  MoveL 9498 to (499.58, 497.3, 18) mm, rotated rx 0 ry 90 rz 0 deg; joints [-11.769, -28.209, 111.796, -15.788, -82.965, 50.97]
  Set speed (15.0 mm/s)
  MoveL 9499 to (498.36, 498.52, 18) mm, rotated rx 0 ry 90 rz 0 deg; joints [-11.905, -28.227, 111.911, -15.921, -83.063, 50.957]
  Set speed (120.0 mm/s)
  MoveL 9500 to (498.02, 497.86, 18) mm, rotated rx 0 ry 90 rz 0 deg; joints [-11.851, -28.235, 111.967, -15.865, -83.107, 50.939]
  Set speed (15.0 mm/s)
  Call Extruder(0.050)
  MoveL 9501 to (499.24, 496.65, 18) mm, rotated rx 0 ry 90 rz 0 deg; joints [-11.715, -28.217, 111.852, -15.733, -83.009, 50.951]
  Set speed (120.0 mm/s)
  MoveL 9502 to (498.91, 495.99, 18) mm, rotated rx 0 ry 90 rz 0 deg; joints [-11.662, -28.226, 111.909, -15.677, -83.053, 50.932]
  Set speed (15.0 mm/s)
  Call Extruder(0.050)
  MoveL 9503 to (497.69, 497.21, 18) mm, rotated rx 0 ry 90 rz 0 deg; joints [-11.797, -28.244, 112.024, -15.81, -83.151, 50.92]
  Set speed (120.0 mm/s)
  MoveL 9504 to (497.36, 496.55, 18) mm, rotated rx 0 ry 90 rz 0 deg; joints [-11.743, -28.253, 112.08, -15.754, -83.195, 50.901]
  Set speed (15.0 mm/s)
  Call Extruder(0.107)
  MoveL 9505 to (499.95, 493.96, 18) mm, rotated rx 0 ry 90 rz 0 deg; joints [-11.455, -28.215, 111.834, -15.471, -82.986, 50.927]
  Set speed (120.0 mm/s)
  MoveL 9506 to (498.96, 493.96, 18) mm, rotated rx 0 ry 90 rz 0 deg; joints [-11.474, -28.233, 111.952, -15.486, -83.083, 50.902]
  Set speed (15.0 mm/s)
  Call Extruder(0.080)
  MoveL 9507 to (497.02, 495.9, 18) mm, rotated rx 0 ry 90 rz 0 deg; joints [-11.689, -28.262, 112.136, -15.698, -83.239, 50.883]
  Set speed (120.0 mm/s)
  MoveL 9508 to (496.69, 495.24, 18) mm, rotated rx 0 ry 90 rz 0 deg; joints [-11.635, -28.27, 112.192, -15.642, -83.283, 50.864]
  Set speed (15.0 mm/s)
  Call Extruder(0.053)
  MoveL 9509 to (497.97, 493.96, 18) mm, rotated rx 0 ry 90 rz 0 deg; joints [-11.492, -28.251, 112.07, -15.502, -83.18, 50.877]
  Set speed (120.0 mm/s)
  MoveL 9510 to (496.98, 493.96, 18) mm, rotated rx 0 ry 90 rz 0 deg; joints [-11.511, -28.27, 112.189, -15.517, -83.277, 50.852]
  Set speed (15.0 mm/s)
  Call Extruder(0.026)
  MoveL 9511 to (496.35, 494.59, 18) mm, rotated rx 0 ry 90 rz 0 deg; joints [-11.58, -28.279, 112.248, -15.586, -83.327, 50.846]
  Set speed (120.0 mm/s)
  MoveL 9512 to (499.33, 495.57, 18) mm, rotated rx 0 ry 90 rz 0 deg; joints [-11.614, -28.22, 111.868, -15.63, -83.019, 50.936]
  Set speed (15.0 mm/s)
  Call Extruder(0.066)
  MoveL 9513 to (500.94, 493.96, 18) mm, rotated rx 0 ry 90 rz 0 deg; joints [-11.437, -28.196, 111.716, -15.456, -82.89, 50.952]
  Set speed (120.0 mm/s)
  MoveL 9514 to (501.93, 493.96, 18) mm, rotated rx 0 ry 90 rz 0 deg; joints [-11.418, -28.177, 111.597, -15.441, -82.793, 50.976]
  Set speed (15.0 mm/s)
  MoveL 9515 to (500.32, 495.57, 18) mm, rotated rx 0 ry 90 rz 0 deg; joints [-11.596, -28.201, 111.75, -15.615, -82.922, 50.961]
  Set speed (120.0 mm/s)
  MoveL 9516 to (501.31, 495.57, 18) mm, rotated rx 0 ry 90 rz 0 deg; joints [-11.577, -28.183, 111.632, -15.599, -82.826, 50.986]
  Set speed (15.0 mm/s)
  MoveL 9517 to (502.92, 493.96, 18) mm, rotated rx 0 ry 90 rz 0 deg; joints [-11.4, -28.158, 111.478, -15.426, -82.697, 51.001]
  Set speed (120.0 mm/s)
  MoveL 9518 to (503.91, 493.96, 18) mm, rotated rx 0 ry 90 rz 0 deg; joints [-11.382, -28.139, 111.36, -15.411, -82.6, 51.026]
  Set speed (15.0 mm/s)
  MoveL 9519 to (502.3, 495.57, 18) mm, rotated rx 0 ry 90 rz 0 deg; joints [-11.558, -28.164, 111.513, -15.584, -82.729, 51.011]
  Set speed (120.0 mm/s)
  MoveL 9520 to (503.29, 495.57, 18) mm, rotated rx 0 ry 90 rz 0 deg; joints [-11.54, -28.144, 111.394, -15.569, -82.633, 51.036]
  Set speed (15.0 mm/s)
  Call Extruder(0.035)
  MoveL 9521 to (504.15, 494.7, 18) mm, rotated rx 0 ry 90 rz 0 deg; joints [-11.445, -28.131, 111.312, -15.476, -82.563, 51.044]
  Set speed (120.0 mm/s)
  MoveL 9522 to (502.26, 502.54, 18) mm, rotated rx 0 ry 90 rz 0 deg; joints [-12.196, -28.136, 111.343, -16.232, -82.613, 51.123]
  Set speed (15.0 mm/s)
  Call Extruder(0.050)
  MoveL 9523 to (501.03, 503.76, 18) mm, rotated rx 0 ry 90 rz 0 deg; joints [-12.332, -28.155, 111.457, -16.365, -82.709, 51.111]
  MoveL 9524 to (500.91, 503.89, 18) mm, rotated rx 0 ry 90 rz 0 deg; joints [-12.346, -28.156, 111.469, -16.379, -82.719, 51.11]
  Set speed (120.0 mm/s)
  MoveL 9525 to (490.68, 490.68, 18) mm, rotated rx 0 ry 90 rz 0 deg; joints [-11.324, -28.393, 113.016, -15.308, -83.95, 50.646]
  Set speed (1000.0 mm/s)
  MoveL 9526 to (490.68, 490.68, 18.1) mm, rotated rx 0 ry 90 rz 0 deg; joints [-11.324, -28.403, 113.021, -15.309, -83.945, 50.647]
  Set speed (30.0 mm/s)
  Call Extruder(0.249)
  MoveL 9527 to (496.74, 496.74, 18.1) mm, rotated rx 0 ry 90 rz 0 deg; joints [-11.772, -28.274, 112.154, -15.781, -83.247, 50.89]
  MoveL 9528 to (496.86, 496.86, 18.1) mm, rotated rx 0 ry 90 rz 0 deg; joints [-11.781, -28.271, 112.137, -15.791, -83.233, 50.895]
  Set speed (120.0 mm/s)
  MoveL 9529 to (495.64, 494.46, 18.1) mm, rotated rx 0 ry 90 rz 0 deg; joints [-11.582, -28.303, 112.341, -15.585, -83.393, 50.827]
  Set speed (30.0 mm/s)
  Call Extruder(0.204)
  MoveL 9530 to (490.68, 499.42, 18.1) mm, rotated rx 0 ry 90 rz 0 deg; joints [-12.139, -28.372, 112.806, -16.133, -83.789, 50.773]
  Set speed (120.0 mm/s)
  MoveL 9531 to (490.68, 500.58, 18.1) mm, rotated rx 0 ry 90 rz 0 deg; joints [-12.247, -28.368, 112.776, -16.242, -83.768, 50.79]
  Set speed (30.0 mm/s)
  Call Extruder(0.208)
  MoveL 9532 to (495.73, 505.63, 18.1) mm, rotated rx 0 ry 90 rz 0 deg; joints [-12.61, -28.257, 112.046, -16.628, -83.184, 51.002]
  Set speed (120.0 mm/s)
  MoveL 9533 to (495.73, 504.27, 18.1) mm, rotated rx 0 ry 90 rz 0 deg; joints [-12.486, -28.263, 112.082, -16.502, -83.209, 50.981]
  Set speed (30.0 mm/s)
  Call Extruder(0.208)
  MoveL 9534 to (490.68, 509.32, 18.1) mm, rotated rx 0 ry 90 rz 0 deg; joints [-13.056, -28.333, 112.544, -17.063, -83.602, 50.924]
  MoveL 9535 to (490.56, 509.44, 18.1) mm, rotated rx 0 ry 90 rz 0 deg; joints [-13.07, -28.335, 112.555, -17.076, -83.611, 50.923]
  Set speed (120.0 mm/s)
  MoveL 9536 to (497.1, 507, 18.1) mm, rotated rx 0 ry 90 rz 0 deg; joints [-12.708, -28.226, 111.846, -16.732, -83.026, 51.062]
  Set speed (30.0 mm/s)
  Call Extruder(0.096)
  MoveL 9537 to (499.42, 509.32, 18.1) mm, rotated rx 0 ry 90 rz 0 deg; joints [-12.872, -28.172, 111.507, -16.907, -82.758, 51.163]
  Set speed (120.0 mm/s)
  MoveL 9538 to (500.58, 509.32, 18.1) mm, rotated rx 0 ry 90 rz 0 deg; joints [-12.847, -28.15, 111.369, -16.888, -82.646, 51.194]
  Set speed (30.0 mm/s)
  Call Extruder(0.096)
  MoveL 9539 to (502.9, 507, 18.1) mm, rotated rx 0 ry 90 rz 0 deg; joints [-12.589, -28.115, 111.153, -16.634, -82.465, 51.216]
  MoveL 9540 to (503.02, 506.87, 18.1) mm, rotated rx 0 ry 90 rz 0 deg; joints [-12.575, -28.113, 111.142, -16.62, -82.455, 51.218]
  Set speed (120.0 mm/s)
  MoveL 9541 to (504.46, 505.44, 18.1) mm, rotated rx 0 ry 90 rz 0 deg; joints [-12.416, -28.091, 111.008, -16.464, -82.343, 51.231]
  Set speed (30.0 mm/s)
  Call Extruder(0.200)
  MoveL 9542 to (509.32, 500.58, 18.1) mm, rotated rx 0 ry 90 rz 0 deg; joints [-11.882, -28.014, 110.549, -15.94, -81.957, 51.273]
  Set speed (120.0 mm/s)
  MoveL 9543 to (509.32, 499.42, 18.1) mm, rotated rx 0 ry 90 rz 0 deg; joints [-11.777, -28.019, 110.579, -15.833, -81.977, 51.253]
  Set speed (30.0 mm/s)
  Call Extruder(0.186)
  MoveL 9544 to (504.79, 494.89, 18.1) mm, rotated rx 0 ry 90 rz 0 deg; joints [-11.45, -28.128, 111.236, -15.484, -82.493, 51.064]
  Set speed (120.0 mm/s)
  MoveL 9545 to (504.79, 495.21, 18.1) mm, rotated rx 0 ry 90 rz 0 deg; joints [-11.479, -28.127, 111.228, -15.513, -82.488, 51.069]
  Set speed (30.0 mm/s)
  Call Extruder(0.186)
  MoveL 9546 to (509.32, 490.68, 18.1) mm, rotated rx 0 ry 90 rz 0 deg; joints [-10.985, -28.055, 110.791, -15.028, -82.12, 51.107]
  MoveL 9547 to (509.44, 490.56, 18.1) mm, rotated rx 0 ry 90 rz 0 deg; joints [-10.972, -28.053, 110.779, -15.015, -82.11, 51.108]
  Set speed (120.0 mm/s)
  MoveL 9548 to (503.23, 493.33, 18.1) mm, rotated rx 0 ry 90 rz 0 deg; joints [-11.336, -28.165, 111.462, -15.362, -82.672, 51]
  Set speed (30.0 mm/s)
  Call Extruder(0.109)
  MoveL 9549 to (500.58, 490.68, 18.1) mm, rotated rx 0 ry 90 rz 0 deg; joints [-11.141, -28.226, 111.842, -15.155, -82.974, 50.894]
  Set speed (120.0 mm/s)
  MoveL 9550 to (499.42, 490.68, 18.1) mm, rotated rx 0 ry 90 rz 0 deg; joints [-11.163, -28.247, 111.981, -15.173, -83.088, 50.865]
  Set speed (30.0 mm/s)
  MoveL 9551 to (496.77, 493.33, 18.1) mm, rotated rx 0 ry 90 rz 0 deg; joints [-11.456, -28.286, 112.233, -15.461, -83.302, 50.839]
  MoveL 9552 to (496.65, 493.45, 18.1) mm, rotated rx 0 ry 90 rz 0 deg; joints [-11.47, -28.288, 112.245, -15.475, -83.312, 50.838]
  Set speed (120.0 mm/s)
  MoveL 9553 to (504.54, 493.58, 18.1) mm, rotated rx 0 ry 90 rz 0 deg; joints [-11.335, -28.138, 111.298, -15.366, -82.539, 51.037]
  Set speed (1000.0 mm/s)
  MoveL 9554 to (504.54, 495.95, 18.1) mm, rotated rx 0 ry 90 rz 0 deg; joints [-11.552, -28.129, 111.24, -15.585, -82.5, 51.075]
  Set speed (1000.0 mm/s)
  MoveL 9555 to (501.11, 498.89, 18.1) mm, rotated rx 0 ry 90 rz 0 deg; joints [-11.886, -28.184, 111.579, -15.912, -82.783, 51.035]
  Set speed (30.0 mm/s)
  Call Extruder(0.111)
  MoveL 9556 to (503.8, 496.2, 18.1) mm, rotated rx 0 ry 90 rz 0 deg; joints [-11.588, -28.143, 111.323, -15.62, -82.568, 51.06]
  MoveL 9557 to (503.92, 496.08, 18.1) mm, rotated rx 0 ry 90 rz 0 deg; joints [-11.575, -28.141, 111.311, -15.607, -82.558, 51.061]
  Set speed (120.0 mm/s)
  MoveL 9558 to (504.54, 493.58, 18.1) mm, rotated rx 0 ry 90 rz 0 deg; joints [-11.335, -28.138, 111.298, -15.366, -82.539, 51.037]
  Set speed (1000.0 mm/s)
  MoveL 9559 to (496.51, 493.57, 18.1) mm, rotated rx 0 ry 90 rz 0 deg; joints [-11.483, -28.29, 112.259, -15.488, -83.324, 50.836]
  Set speed (1000.0 mm/s)
  MoveL 9560 to (498.94, 501.06, 18.1) mm, rotated rx 0 ry 90 rz 0 deg; joints [-12.126, -28.216, 111.782, -16.149, -82.956, 51.014]
  Set speed (30.0 mm/s)
  Call Extruder(0.126)
  MoveL 9561 to (495.87, 504.12, 18.1) mm, rotated rx 0 ry 90 rz 0 deg; joints [-12.469, -28.261, 112.068, -16.486, -83.197, 50.982]
  MoveL 9562 to (495.75, 504.25, 18.1) mm, rotated rx 0 ry 90 rz 0 deg; joints [-12.483, -28.263, 112.079, -16.499, -83.207, 50.981]
  Set speed (120.0 mm/s)
  MoveL 9563 to (495.98, 506.75, 18.1) mm, rotated rx 0 ry 90 rz 0 deg; joints [-12.708, -28.248, 111.986, -16.728, -83.139, 51.027]
  Set speed (1000.0 mm/s)
  MoveL 9564 to (504.36, 506.75, 18.1) mm, rotated rx 0 ry 90 rz 0 deg; joints [-12.537, -28.087, 110.986, -16.586, -82.329, 51.251]
  Set speed (1000.0 mm/s)
  MoveL 9565 to (503.43, 503.43, 18.1) mm, rotated rx 0 ry 90 rz 0 deg; joints [-12.254, -28.12, 111.185, -16.295, -82.478, 51.17]
  Set speed (30.0 mm/s)
  Call Extruder(0.243)
  MoveL 9566 to (509.32, 509.32, 18.1) mm, rotated rx 0 ry 90 rz 0 deg; joints [-12.669, -27.974, 110.32, -16.742, -81.804, 51.427]
  MoveL 9567 to (509.44, 509.44, 18.1) mm, rotated rx 0 ry 90 rz 0 deg; joints [-12.677, -27.971, 110.302, -16.751, -81.79, 51.433]
  Set speed (120.0 mm/s)
  MoveL 9568 to (495.98, 506.75, 18.1) mm, rotated rx 0 ry 90 rz 0 deg; joints [-12.708, -28.248, 111.986, -16.728, -83.139, 51.027]
  Set speed (1000.0 mm/s)
  MoveL 9569 to (495.94, 504.33, 18.1) mm, rotated rx 0 ry 90 rz 0 deg; joints [-12.487, -28.259, 112.055, -16.504, -83.188, 50.987]
  Set speed (1000.0 mm/s)
  MoveL 9570 to (496.01, 504.41, 18.1) mm, rotated rx 0 ry 90 rz 0 deg; joints [-12.492, -28.257, 112.045, -16.509, -83.179, 50.99]
  Set speed (15.0 mm/s)
  Call Extruder(0.067)
  MoveL 9571 to (496.01, 506.72, 18.1) mm, rotated rx 0 ry 90 rz 0 deg; joints [-12.705, -28.248, 111.983, -16.725, -83.136, 51.028]
  Call Extruder(0.242)
  MoveL 9572 to (504.33, 506.72, 18.1) mm, rotated rx 0 ry 90 rz 0 deg; joints [-12.535, -28.088, 110.99, -16.584, -82.332, 51.249]
  Call Extruder(0.027)
  MoveL 9573 to (504.33, 505.8, 18.1) mm, rotated rx 0 ry 90 rz 0 deg; joints [-12.452, -28.092, 111.014, -16.5, -82.349, 51.234]
  Call Extruder(0.306)
  MoveL 9574 to (499.53, 496.43, 18.1) mm, rotated rx 0 ry 90 rz 0 deg; joints [-11.69, -28.223, 111.829, -15.708, -82.98, 50.956]
  Call Extruder(0.017)
  MoveL 9575 to (499.27, 495.92, 18.1) mm, rotated rx 0 ry 90 rz 0 deg; joints [-11.648, -28.23, 111.872, -15.665, -83.014, 50.942]
  Call Extruder(0.010)
  MoveL 9576 to (499.84, 495.92, 18.1) mm, rotated rx 0 ry 90 rz 0 deg; joints [-11.637, -28.22, 111.804, -15.656, -82.958, 50.956]
  Call Extruder(0.000)
  MoveL 9577 to (499.84, 495.92, 18.1) mm, rotated rx 0 ry 90 rz 0 deg; joints [-11.637, -28.22, 111.804, -15.656, -82.958, 50.956]
  Call Extruder(0.136)
  MoveL 9578 to (504.51, 495.92, 18.1) mm, rotated rx 0 ry 90 rz 0 deg; joints [-11.55, -28.13, 111.244, -15.583, -82.503, 51.074]
  Call Extruder(0.067)
  MoveL 9579 to (504.51, 493.61, 18.1) mm, rotated rx 0 ry 90 rz 0 deg; joints [-11.338, -28.139, 111.301, -15.369, -82.542, 51.037]
  Call Extruder(0.233)
  MoveL 9580 to (496.51, 493.61, 18.1) mm, rotated rx 0 ry 90 rz 0 deg; joints [-11.487, -28.29, 112.258, -15.492, -83.323, 50.837]
  Call Extruder(0.017)
  MoveL 9581 to (495.92, 493.64, 18.1) mm, rotated rx 0 ry 90 rz 0 deg; joints [-11.501, -28.301, 112.327, -15.504, -83.38, 50.822]
  Call Extruder(0.026)
  MoveL 9582 to (495.92, 494.52, 18.1) mm, rotated rx 0 ry 90 rz 0 deg; joints [-11.583, -28.297, 112.306, -15.587, -83.365, 50.835]
  Call Extruder(0.306)
  MoveL 9583 to (500.7, 503.9, 18.1) mm, rotated rx 0 ry 90 rz 0 deg; joints [-12.351, -28.171, 111.498, -16.383, -82.734, 51.106]
  Call Extruder(0.017)
  MoveL 9584 to (500.96, 504.4, 18.1) mm, rotated rx 0 ry 90 rz 0 deg; joints [-12.392, -28.164, 111.454, -16.426, -82.699, 51.122]
  Call Extruder(0.010)
  MoveL 9585 to (500.39, 504.41, 18.1) mm, rotated rx 0 ry 90 rz 0 deg; joints [-12.404, -28.175, 111.522, -16.436, -82.754, 51.107]
  Call Extruder(0.000)
  MoveL 9586 to (500.39, 504.41, 18.1) mm, rotated rx 0 ry 90 rz 0 deg; joints [-12.404, -28.175, 111.522, -16.436, -82.755, 51.107]
  Call Extruder(0.128)
  MoveL 9587 to (496.01, 504.41, 18.1) mm, rotated rx 0 ry 90 rz 0 deg; joints [-12.492, -28.257, 112.045, -16.509, -83.179, 50.99]
  Set speed (120.0 mm/s)
  MoveL 9588 to (496.01, 504.81, 18.1) mm, rotated rx 0 ry 90 rz 0 deg; joints [-12.529, -28.256, 112.034, -16.547, -83.172, 50.997]
  Set speed (1000.0 mm/s)
  MoveL 9589 to (495.91, 504.81, 18.1) mm, rotated rx 0 ry 90 rz 0 deg; joints [-12.531, -28.257, 112.046, -16.548, -83.182, 50.994]
  Set speed (1000.0 mm/s)
  MoveL 9590 to (490.47, 509.53, 18.1) mm, rotated rx 0 ry 90 rz 0 deg; joints [-13.08, -28.336, 112.563, -17.086, -83.618, 50.922]
  Set speed (1000.0 mm/s)
  MoveL 9591 to (490.4, 509.6, 18.1) mm, rotated rx 0 ry 90 rz 0 deg; joints [-13.088, -28.337, 112.569, -17.094, -83.623, 50.921]
  Set speed (15.0 mm/s)
  Call Extruder(0.559)
  MoveL 9592 to (490.4, 490.4, 18.1) mm, rotated rx 0 ry 90 rz 0 deg; joints [-11.303, -28.409, 113.06, -15.287, -83.977, 50.636]
  MoveL 9593 to (509.6, 490.4, 18.1) mm, rotated rx 0 ry 90 rz 0 deg; joints [-10.955, -28.05, 110.764, -14.998, -82.097, 51.109]
  MoveL 9594 to (509.6, 509.6, 18.1) mm, rotated rx 0 ry 90 rz 0 deg; joints [-12.688, -27.967, 110.278, -16.763, -81.772, 51.44]
  MoveL 9595 to (490.4, 509.6, 18.1) mm, rotated rx 0 ry 90 rz 0 deg; joints [-13.088, -28.337, 112.569, -17.094, -83.623, 50.921]
  Set speed (120.0 mm/s)
  MoveL 9596 to (490.4, 509.2, 18.1) mm, rotated rx 0 ry 90 rz 0 deg; joints [-13.051, -28.339, 112.58, -17.056, -83.631, 50.915]
  Set speed (1000.0 mm/s)
  MoveL 9597 to (491.1, 508.9, 18.1) mm, rotated rx 0 ry 90 rz 0 deg; joints [-13.008, -28.328, 112.506, -17.016, -83.569, 50.929]
  Set speed (1000.0 mm/s)
  MoveL 9598 to (490.68, 490.68, 18.1) mm, rotated rx 0 ry 90 rz 0 deg; joints [-11.324, -28.403, 113.021, -15.309, -83.945, 50.647]
  Set speed (1000.0 mm/s)
  MoveL 9599 to (490.68, 490.68, 18.2) mm, rotated rx 0 ry 90 rz 0 deg; joints [-11.324, -28.414, 113.026, -15.309, -83.939, 50.649]
  Set speed (30.0 mm/s)
  Call Extruder(0.249)
  MoveL 9600 to (496.74, 496.74, 18.2) mm, rotated rx 0 ry 90 rz 0 deg; joints [-11.772, -28.285, 112.159, -15.781, -83.241, 50.891]
  MoveL 9601 to (496.86, 496.86, 18.2) mm, rotated rx 0 ry 90 rz 0 deg; joints [-11.781, -28.282, 112.142, -15.791, -83.227, 50.896]
  Set speed (120.0 mm/s)
  MoveL 9602 to (495.64, 494.46, 18.2) mm, rotated rx 0 ry 90 rz 0 deg; joints [-11.582, -28.313, 112.346, -15.585, -83.388, 50.829]
  Set speed (30.0 mm/s)
  Call Extruder(0.204)
  MoveL 9603 to (490.68, 499.42, 18.2) mm, rotated rx 0 ry 90 rz 0 deg; joints [-12.139, -28.383, 112.811, -16.133, -83.784, 50.774]
  Set speed (120.0 mm/s)
  MoveL 9604 to (490.68, 500.58, 18.2) mm, rotated rx 0 ry 90 rz 0 deg; joints [-12.247, -28.378, 112.781, -16.243, -83.763, 50.791]
  Set speed (30.0 mm/s)
  Call Extruder(0.208)
  MoveL 9605 to (495.73, 505.63, 18.2) mm, rotated rx 0 ry 90 rz 0 deg; joints [-12.61, -28.268, 112.051, -16.628, -83.179, 51.004]
  Set speed (120.0 mm/s)
  MoveL 9606 to (495.73, 504.27, 18.2) mm, rotated rx 0 ry 90 rz 0 deg; joints [-12.486, -28.274, 112.087, -16.502, -83.204, 50.982]
  Set speed (30.0 mm/s)
  Call Extruder(0.208)
  MoveL 9607 to (490.68, 509.32, 18.2) mm, rotated rx 0 ry 90 rz 0 deg; joints [-13.056, -28.344, 112.549, -17.063, -83.596, 50.926]
  MoveL 9608 to (490.56, 509.44, 18.2) mm, rotated rx 0 ry 90 rz 0 deg; joints [-13.07, -28.346, 112.56, -17.076, -83.606, 50.924]
  Set speed (120.0 mm/s)
  MoveL 9609 to (497.1, 507, 18.2) mm, rotated rx 0 ry 90 rz 0 deg; joints [-12.708, -28.237, 111.851, -16.732, -83.02, 51.063]
  Set speed (30.0 mm/s)
  Call Extruder(0.096)
  MoveL 9610 to (499.42, 509.32, 18.2) mm, rotated rx 0 ry 90 rz 0 deg; joints [-12.872, -28.183, 111.512, -16.908, -82.752, 51.164]
  Set speed (120.0 mm/s)
  MoveL 9611 to (500.58, 509.32, 18.2) mm, rotated rx 0 ry 90 rz 0 deg; joints [-12.847, -28.161, 111.374, -16.888, -82.641, 51.196]
  Set speed (30.0 mm/s)
  Call Extruder(0.096)
  MoveL 9612 to (502.9, 507, 18.2) mm, rotated rx 0 ry 90 rz 0 deg; joints [-12.589, -28.125, 111.159, -16.634, -82.459, 51.218]
  MoveL 9613 to (503.02, 506.87, 18.2) mm, rotated rx 0 ry 90 rz 0 deg; joints [-12.575, -28.123, 111.147, -16.62, -82.45, 51.219]
  Set speed (120.0 mm/s)
  MoveL 9614 to (504.46, 505.44, 18.2) mm, rotated rx 0 ry 90 rz 0 deg; joints [-12.416, -28.101, 111.013, -16.465, -82.337, 51.232]
  Set speed (30.0 mm/s)
  Call Extruder(0.200)
  MoveL 9615 to (509.32, 500.58, 18.2) mm, rotated rx 0 ry 90 rz 0 deg; joints [-11.882, -28.024, 110.554, -15.94, -81.952, 51.274]
  Set speed (120.0 mm/s)
  MoveL 9616 to (509.32, 499.42, 18.2) mm, rotated rx 0 ry 90 rz 0 deg; joints [-11.777, -28.029, 110.584, -15.834, -81.971, 51.254]
  Set speed (30.0 mm/s)
  Call Extruder(0.186)
  MoveL 9617 to (504.79, 494.89, 18.2) mm, rotated rx 0 ry 90 rz 0 deg; joints [-11.45, -28.139, 111.241, -15.484, -82.488, 51.066]
  Set speed (120.0 mm/s)
  MoveL 9618 to (504.79, 495.21, 18.2) mm, rotated rx 0 ry 90 rz 0 deg; joints [-11.479, -28.138, 111.233, -15.513, -82.482, 51.071]
  Set speed (30.0 mm/s)
  Call Extruder(0.186)
  MoveL 9619 to (509.32, 490.68, 18.2) mm, rotated rx 0 ry 90 rz 0 deg; joints [-10.985, -28.065, 110.796, -15.028, -82.115, 51.108]
  MoveL 9620 to (509.44, 490.56, 18.2) mm, rotated rx 0 ry 90 rz 0 deg; joints [-10.972, -28.063, 110.784, -15.015, -82.105, 51.109]
  Set speed (120.0 mm/s)
  MoveL 9621 to (503.23, 493.33, 18.2) mm, rotated rx 0 ry 90 rz 0 deg; joints [-11.336, -28.176, 111.467, -15.362, -82.666, 51.002]
  Set speed (30.0 mm/s)
  Call Extruder(0.109)
  MoveL 9622 to (500.58, 490.68, 18.2) mm, rotated rx 0 ry 90 rz 0 deg; joints [-11.141, -28.236, 111.847, -15.155, -82.969, 50.895]
  Set speed (120.0 mm/s)
  MoveL 9623 to (499.42, 490.68, 18.2) mm, rotated rx 0 ry 90 rz 0 deg; joints [-11.163, -28.258, 111.986, -15.173, -83.083, 50.867]
  Set speed (30.0 mm/s)
  MoveL 9624 to (496.77, 493.33, 18.2) mm, rotated rx 0 ry 90 rz 0 deg; joints [-11.456, -28.297, 112.238, -15.462, -83.297, 50.841]
  MoveL 9625 to (496.65, 493.45, 18.2) mm, rotated rx 0 ry 90 rz 0 deg; joints [-11.47, -28.299, 112.25, -15.475, -83.307, 50.839]
  Set speed (120.0 mm/s)
  MoveL 9626 to (504.54, 493.58, 18.2) mm, rotated rx 0 ry 90 rz 0 deg; joints [-11.335, -28.149, 111.303, -15.366, -82.534, 51.038]
  Set speed (1000.0 mm/s)
  MoveL 9627 to (504.54, 495.95, 18.2) mm, rotated rx 0 ry 90 rz 0 deg; joints [-11.552, -28.14, 111.245, -15.586, -82.494, 51.076]
  Set speed (1000.0 mm/s)
  MoveL 9628 to (501.11, 498.89, 18.2) mm, rotated rx 0 ry 90 rz 0 deg; joints [-11.886, -28.194, 111.584, -15.912, -82.778, 51.037]
  Set speed (30.0 mm/s)
  Call Extruder(0.111)
  MoveL 9629 to (503.8, 496.2, 18.2) mm, rotated rx 0 ry 90 rz 0 deg; joints [-11.588, -28.153, 111.328, -15.62, -82.562, 51.062]
  MoveL 9630 to (503.92, 496.08, 18.2) mm, rotated rx 0 ry 90 rz 0 deg; joints [-11.575, -28.151, 111.316, -15.607, -82.553, 51.063]
  Set speed (120.0 mm/s)
  MoveL 9631 to (504.54, 493.58, 18.2) mm, rotated rx 0 ry 90 rz 0 deg; joints [-11.335, -28.149, 111.303, -15.366, -82.534, 51.038]
  Set speed (1000.0 mm/s)
  MoveL 9632 to (495.89, 493.58, 18.2) mm, rotated rx 0 ry 90 rz 0 deg; joints [-11.496, -28.312, 112.337, -15.499, -83.378, 50.822]
  Set speed (1000.0 mm/s)
  MoveL 9633 to (498.94, 501.06, 18.2) mm, rotated rx 0 ry 90 rz 0 deg; joints [-12.126, -28.227, 111.787, -16.149, -82.95, 51.016]
  Set speed (30.0 mm/s)
  Call Extruder(0.126)
  MoveL 9634 to (495.87, 504.12, 18.2) mm, rotated rx 0 ry 90 rz 0 deg; joints [-12.469, -28.271, 112.073, -16.486, -83.192, 50.984]
  MoveL 9635 to (495.75, 504.25, 18.2) mm, rotated rx 0 ry 90 rz 0 deg; joints [-12.483, -28.273, 112.084, -16.499, -83.202, 50.983]
  Set speed (120.0 mm/s)
  MoveL 9636 to (495.98, 506.75, 18.2) mm, rotated rx 0 ry 90 rz 0 deg; joints [-12.708, -28.259, 111.991, -16.728, -83.133, 51.029]
  Set speed (1000.0 mm/s)
  MoveL 9637 to (504.36, 506.75, 18.2) mm, rotated rx 0 ry 90 rz 0 deg; joints [-12.537, -28.098, 110.991, -16.587, -82.324, 51.252]
  Set speed (1000.0 mm/s)
  MoveL 9638 to (503.43, 503.43, 18.2) mm, rotated rx 0 ry 90 rz 0 deg; joints [-12.254, -28.131, 111.19, -16.295, -82.473, 51.171]
  Set speed (30.0 mm/s)
  Call Extruder(0.243)
  MoveL 9639 to (509.32, 509.32, 18.2) mm, rotated rx 0 ry 90 rz 0 deg; joints [-12.669, -27.985, 110.325, -16.742, -81.799, 51.429]
  MoveL 9640 to (509.44, 509.44, 18.2) mm, rotated rx 0 ry 90 rz 0 deg; joints [-12.677, -27.982, 110.307, -16.751, -81.785, 51.434]
  Set speed (120.0 mm/s)
  MoveL 9641 to (495.98, 506.75, 18.2) mm, rotated rx 0 ry 90 rz 0 deg; joints [-12.708, -28.259, 111.991, -16.728, -83.133, 51.029]
  Set speed (1000.0 mm/s)
  MoveL 9642 to (495.94, 504.34, 18.2) mm, rotated rx 0 ry 90 rz 0 deg; joints [-12.487, -28.269, 112.06, -16.504, -83.182, 50.989]
  Set speed (1000.0 mm/s)
  MoveL 9643 to (496.01, 504.41, 18.2) mm, rotated rx 0 ry 90 rz 0 deg; joints [-12.492, -28.268, 112.05, -16.51, -83.174, 50.992]
  Set speed (15.0 mm/s)
  Call Extruder(0.067)
  MoveL 9644 to (496.01, 506.72, 18.2) mm, rotated rx 0 ry 90 rz 0 deg; joints [-12.705, -28.258, 111.989, -16.725, -83.131, 51.029]
  Call Extruder(0.242)
  MoveL 9645 to (504.33, 506.72, 18.2) mm, rotated rx 0 ry 90 rz 0 deg; joints [-12.535, -28.098, 110.995, -16.585, -82.327, 51.251]
  Call Extruder(0.027)
  MoveL 9646 to (504.33, 505.8, 18.2) mm, rotated rx 0 ry 90 rz 0 deg; joints [-12.452, -28.102, 111.019, -16.5, -82.343, 51.235]
  Call Extruder(0.306)
  MoveL 9647 to (499.53, 496.43, 18.2) mm, rotated rx 0 ry 90 rz 0 deg; joints [-11.69, -28.234, 111.834, -15.708, -82.974, 50.958]
  Call Extruder(0.017)
  MoveL 9648 to (499.27, 495.92, 18.2) mm, rotated rx 0 ry 90 rz 0 deg; joints [-11.648, -28.241, 111.877, -15.665, -83.008, 50.943]
  Call Extruder(0.010)
  MoveL 9649 to (499.84, 495.92, 18.2) mm, rotated rx 0 ry 90 rz 0 deg; joints [-11.637, -28.23, 111.809, -15.656, -82.953, 50.958]
  Call Extruder(0.000)
  MoveL 9650 to (499.84, 495.92, 18.2) mm, rotated rx 0 ry 90 rz 0 deg; joints [-11.637, -28.23, 111.809, -15.656, -82.953, 50.958]
  Call Extruder(0.136)
  MoveL 9651 to (504.51, 495.92, 18.2) mm, rotated rx 0 ry 90 rz 0 deg; joints [-11.55, -28.14, 111.249, -15.583, -82.498, 51.075]
  Call Extruder(0.067)
  MoveL 9652 to (504.51, 493.61, 18.2) mm, rotated rx 0 ry 90 rz 0 deg; joints [-11.338, -28.149, 111.306, -15.369, -82.536, 51.038]
  Call Extruder(0.250)
  MoveL 9653 to (495.92, 493.61, 18.2) mm, rotated rx 0 ry 90 rz 0 deg; joints [-11.498, -28.311, 112.333, -15.501, -83.375, 50.823]
  Call Extruder(0.027)
  MoveL 9654 to (495.92, 494.52, 18.2) mm, rotated rx 0 ry 90 rz 0 deg; joints [-11.583, -28.308, 112.311, -15.587, -83.359, 50.837]
  Call Extruder(0.306)
  MoveL 9655 to (500.7, 503.9, 18.2) mm, rotated rx 0 ry 90 rz 0 deg; joints [-12.351, -28.181, 111.503, -16.384, -82.728, 51.108]
  Call Extruder(0.017)
  MoveL 9656 to (500.96, 504.41, 18.2) mm, rotated rx 0 ry 90 rz 0 deg; joints [-12.392, -28.174, 111.459, -16.426, -82.694, 51.123]
  Call Extruder(0.010)
  MoveL 9657 to (500.39, 504.4, 18.2) mm, rotated rx 0 ry 90 rz 0 deg; joints [-12.404, -28.185, 111.527, -16.436, -82.749, 51.108]
  Call Extruder(0.000)
  MoveL 9658 to (500.39, 504.41, 18.2) mm, rotated rx 0 ry 90 rz 0 deg; joints [-12.404, -28.185, 111.527, -16.436, -82.749, 51.108]
  Call Extruder(0.128)
  MoveL 9659 to (496.01, 504.41, 18.2) mm, rotated rx 0 ry 90 rz 0 deg; joints [-12.492, -28.268, 112.05, -16.51, -83.174, 50.992]
  Set speed (120.0 mm/s)
  MoveL 9660 to (496.01, 504.81, 18.2) mm, rotated rx 0 ry 90 rz 0 deg; joints [-12.529, -28.266, 112.039, -16.547, -83.167, 50.998]
  Set speed (1000.0 mm/s)
  MoveL 9661 to (495.91, 504.8, 18.2) mm, rotated rx 0 ry 90 rz 0 deg; joints [-12.531, -28.268, 112.051, -16.549, -83.176, 50.996]
  Set speed (1000.0 mm/s)
  MoveL 9662 to (490.47, 509.53, 18.2) mm, rotated rx 0 ry 90 rz 0 deg; joints [-13.08, -28.347, 112.568, -17.086, -83.612, 50.923]
  Set speed (1000.0 mm/s)
  MoveL 9663 to (490.4, 509.6, 18.2) mm, rotated rx 0 ry 90 rz 0 deg; joints [-13.088, -28.348, 112.575, -17.094, -83.618, 50.923]
  Set speed (15.0 mm/s)
  Call Extruder(0.559)
  MoveL 9664 to (490.4, 490.4, 18.2) mm, rotated rx 0 ry 90 rz 0 deg; joints [-11.303, -28.42, 113.065, -15.287, -83.972, 50.638]
  MoveL 9665 to (509.6, 490.4, 18.2) mm, rotated rx 0 ry 90 rz 0 deg; joints [-10.955, -28.06, 110.769, -14.998, -82.092, 51.111]
  MoveL 9666 to (509.6, 509.6, 18.2) mm, rotated rx 0 ry 90 rz 0 deg; joints [-12.688, -27.978, 110.283, -16.763, -81.766, 51.441]
  MoveL 9667 to (490.4, 509.6, 18.2) mm, rotated rx 0 ry 90 rz 0 deg; joints [-13.088, -28.348, 112.575, -17.094, -83.618, 50.923]
  Set speed (120.0 mm/s)
  MoveL 9668 to (490.4, 509.2, 18.2) mm, rotated rx 0 ry 90 rz 0 deg; joints [-13.051, -28.349, 112.586, -17.057, -83.626, 50.916]
  Set speed (1000.0 mm/s)
  MoveL 9669 to (491.1, 508.9, 18.2) mm, rotated rx 0 ry 90 rz 0 deg; joints [-13.008, -28.338, 112.511, -17.016, -83.564, 50.931]
  Set speed (1000.0 mm/s)
  MoveL 9670 to (490.68, 490.68, 18.2) mm, rotated rx 0 ry 90 rz 0 deg; joints [-11.324, -28.414, 113.026, -15.309, -83.939, 50.649]
  Set speed (1000.0 mm/s)
  MoveL 9671 to (490.68, 490.68, 18.3) mm, rotated rx 0 ry 90 rz 0 deg; joints [-11.324, -28.425, 113.031, -15.309, -83.934, 50.65]
  Set speed (30.0 mm/s)
  Call Extruder(0.249)
  MoveL 9672 to (496.74, 496.74, 18.3) mm, rotated rx 0 ry 90 rz 0 deg; joints [-11.772, -28.295, 112.164, -15.781, -83.236, 50.893]
  MoveL 9673 to (496.86, 496.86, 18.3) mm, rotated rx 0 ry 90 rz 0 deg; joints [-11.781, -28.293, 112.147, -15.791, -83.222, 50.898]
  Set speed (120.0 mm/s)
  MoveL 9674 to (495.64, 494.46, 18.3) mm, rotated rx 0 ry 90 rz 0 deg; joints [-11.582, -28.324, 112.351, -15.586, -83.383, 50.83]
  Set speed (30.0 mm/s)
  Call Extruder(0.204)
  MoveL 9675 to (490.68, 499.42, 18.3) mm, rotated rx 0 ry 90 rz 0 deg; joints [-12.139, -28.393, 112.816, -16.134, -83.779, 50.776]
  Set speed (120.0 mm/s)
  MoveL 9676 to (490.68, 500.58, 18.3) mm, rotated rx 0 ry 90 rz 0 deg; joints [-12.247, -28.389, 112.786, -16.243, -83.757, 50.793]
  Set speed (30.0 mm/s)
  Call Extruder(0.208)
  MoveL 9677 to (495.73, 505.63, 18.3) mm, rotated rx 0 ry 90 rz 0 deg; joints [-12.61, -28.279, 112.056, -16.628, -83.173, 51.006]
  Set speed (120.0 mm/s)
  MoveL 9678 to (495.72, 504.27, 18.3) mm, rotated rx 0 ry 90 rz 0 deg; joints [-12.486, -28.284, 112.092, -16.502, -83.199, 50.984]
  Set speed (30.0 mm/s)
  Call Extruder(0.208)
  MoveL 9679 to (490.68, 509.32, 18.3) mm, rotated rx 0 ry 90 rz 0 deg; joints [-13.056, -28.355, 112.554, -17.063, -83.591, 50.927]
  MoveL 9680 to (490.56, 509.44, 18.3) mm, rotated rx 0 ry 90 rz 0 deg; joints [-13.07, -28.356, 112.566, -17.077, -83.601, 50.926]
  Set speed (120.0 mm/s)
  MoveL 9681 to (497.1, 507, 18.3) mm, rotated rx 0 ry 90 rz 0 deg; joints [-12.708, -28.247, 111.856, -16.732, -83.015, 51.065]
  Set speed (30.0 mm/s)
  Call Extruder(0.096)
  MoveL 9682 to (499.42, 509.32, 18.3) mm, rotated rx 0 ry 90 rz 0 deg; joints [-12.872, -28.193, 111.517, -16.908, -82.747, 51.166]
  Set speed (120.0 mm/s)
  MoveL 9683 to (500.58, 509.32, 18.3) mm, rotated rx 0 ry 90 rz 0 deg; joints [-12.847, -28.171, 111.379, -16.888, -82.635, 51.197]
  Set speed (30.0 mm/s)
  Call Extruder(0.096)
  MoveL 9684 to (502.9, 507, 18.3) mm, rotated rx 0 ry 90 rz 0 deg; joints [-12.589, -28.136, 111.164, -16.634, -82.454, 51.22]
  MoveL 9685 to (503.02, 506.87, 18.3) mm, rotated rx 0 ry 90 rz 0 deg; joints [-12.575, -28.134, 111.152, -16.621, -82.445, 51.221]
  Set speed (120.0 mm/s)
  MoveL 9686 to (504.46, 505.44, 18.3) mm, rotated rx 0 ry 90 rz 0 deg; joints [-12.416, -28.112, 111.018, -16.465, -82.332, 51.234]
  Set speed (30.0 mm/s)
  Call Extruder(0.200)
  MoveL 9687 to (509.32, 500.58, 18.3) mm, rotated rx 0 ry 90 rz 0 deg; joints [-11.882, -28.035, 110.559, -15.94, -81.947, 51.276]
  Set speed (120.0 mm/s)
  MoveL 9688 to (509.32, 499.42, 18.3) mm, rotated rx 0 ry 90 rz 0 deg; joints [-11.777, -28.04, 110.589, -15.834, -81.966, 51.256]
  Set speed (30.0 mm/s)
  Call Extruder(0.186)
  MoveL 9689 to (504.79, 494.89, 18.3) mm, rotated rx 0 ry 90 rz 0 deg; joints [-11.45, -28.149, 111.246, -15.484, -82.483, 51.067]
  Set speed (120.0 mm/s)
  MoveL 9690 to (504.79, 495.21, 18.3) mm, rotated rx 0 ry 90 rz 0 deg; joints [-11.479, -28.148, 111.238, -15.513, -82.477, 51.072]
  Set speed (30.0 mm/s)
  Call Extruder(0.186)
  MoveL 9691 to (509.32, 490.68, 18.3) mm, rotated rx 0 ry 90 rz 0 deg; joints [-10.985, -28.076, 110.801, -15.028, -82.109, 51.11]
  MoveL 9692 to (509.44, 490.56, 18.3) mm, rotated rx 0 ry 90 rz 0 deg; joints [-10.972, -28.074, 110.789, -15.015, -82.099, 51.111]
  Set speed (120.0 mm/s)
  MoveL 9693 to (503.23, 493.33, 18.3) mm, rotated rx 0 ry 90 rz 0 deg; joints [-11.336, -28.186, 111.472, -15.362, -82.661, 51.003]
  Set speed (30.0 mm/s)
  Call Extruder(0.109)
  MoveL 9694 to (500.58, 490.68, 18.3) mm, rotated rx 0 ry 90 rz 0 deg; joints [-11.141, -28.247, 111.852, -15.156, -82.964, 50.897]
  Set speed (120.0 mm/s)
  MoveL 9695 to (499.42, 490.68, 18.3) mm, rotated rx 0 ry 90 rz 0 deg; joints [-11.163, -28.268, 111.991, -15.173, -83.077, 50.868]
  Set speed (30.0 mm/s)
  MoveL 9696 to (496.77, 493.33, 18.3) mm, rotated rx 0 ry 90 rz 0 deg; joints [-11.456, -28.308, 112.244, -15.462, -83.292, 50.842]
  MoveL 9697 to (496.65, 493.45, 18.3) mm, rotated rx 0 ry 90 rz 0 deg; joints [-11.47, -28.309, 112.255, -15.475, -83.302, 50.841]
  Set speed (120.0 mm/s)
  MoveL 9698 to (504.54, 493.58, 18.3) mm, rotated rx 0 ry 90 rz 0 deg; joints [-11.335, -28.16, 111.308, -15.366, -82.529, 51.04]
  Set speed (1000.0 mm/s)
  MoveL 9699 to (504.54, 495.95, 18.3) mm, rotated rx 0 ry 90 rz 0 deg; joints [-11.552, -28.15, 111.25, -15.586, -82.489, 51.078]
  Set speed (1000.0 mm/s)
  MoveL 9700 to (501.11, 498.89, 18.3) mm, rotated rx 0 ry 90 rz 0 deg; joints [-11.886, -28.205, 111.589, -15.913, -82.773, 51.038]
  Set speed (30.0 mm/s)
  Call Extruder(0.111)
  MoveL 9701 to (503.8, 496.2, 18.3) mm, rotated rx 0 ry 90 rz 0 deg; joints [-11.588, -28.164, 111.333, -15.621, -82.557, 51.063]
  MoveL 9702 to (503.92, 496.08, 18.3) mm, rotated rx 0 ry 90 rz 0 deg; joints [-11.575, -28.162, 111.321, -15.607, -82.547, 51.064]
  Set speed (120.0 mm/s)
  MoveL 9703 to (504.54, 493.58, 18.3) mm, rotated rx 0 ry 90 rz 0 deg; joints [-11.335, -28.16, 111.308, -15.366, -82.529, 51.04]
  Set speed (1000.0 mm/s)
  MoveL 9704 to (495.89, 493.58, 18.3) mm, rotated rx 0 ry 90 rz 0 deg; joints [-11.496, -28.323, 112.342, -15.499, -83.373, 50.824]
  Set speed (1000.0 mm/s)
  MoveL 9705 to (498.94, 501.06, 18.3) mm, rotated rx 0 ry 90 rz 0 deg; joints [-12.126, -28.237, 111.793, -16.149, -82.945, 51.017]
  Set speed (30.0 mm/s)
  Call Extruder(0.126)
  MoveL 9706 to (495.87, 504.12, 18.3) mm, rotated rx 0 ry 90 rz 0 deg; joints [-12.469, -28.282, 112.078, -16.486, -83.187, 50.986]
  MoveL 9707 to (495.75, 504.25, 18.3) mm, rotated rx 0 ry 90 rz 0 deg; joints [-12.483, -28.284, 112.09, -16.499, -83.197, 50.984]
  Set speed (120.0 mm/s)
  MoveL 9708 to (495.98, 506.75, 18.3) mm, rotated rx 0 ry 90 rz 0 deg; joints [-12.708, -28.269, 111.996, -16.728, -83.128, 51.031]
  Set speed (1000.0 mm/s)
  MoveL 9709 to (504.36, 506.75, 18.3) mm, rotated rx 0 ry 90 rz 0 deg; joints [-12.537, -28.108, 110.996, -16.587, -82.318, 51.254]
  Set speed (1000.0 mm/s)
  MoveL 9710 to (503.43, 503.43, 18.3) mm, rotated rx 0 ry 90 rz 0 deg; joints [-12.254, -28.141, 111.195, -16.296, -82.468, 51.173]
  Set speed (30.0 mm/s)
  Call Extruder(0.243)
  MoveL 9711 to (509.32, 509.32, 18.3) mm, rotated rx 0 ry 90 rz 0 deg; joints [-12.669, -27.995, 110.33, -16.742, -81.793, 51.43]
  MoveL 9712 to (509.44, 509.44, 18.3) mm, rotated rx 0 ry 90 rz 0 deg; joints [-12.677, -27.992, 110.312, -16.751, -81.779, 51.436]
  Set speed (120.0 mm/s)
  MoveL 9713 to (495.98, 506.75, 18.3) mm, rotated rx 0 ry 90 rz 0 deg; joints [-12.708, -28.269, 111.996, -16.728, -83.128, 51.031]
  Set speed (1000.0 mm/s)
  MoveL 9714 to (495.94, 504.33, 18.3) mm, rotated rx 0 ry 90 rz 0 deg; joints [-12.487, -28.28, 112.065, -16.505, -83.177, 50.991]
  Set speed (1000.0 mm/s)
  MoveL 9715 to (496.01, 504.41, 18.3) mm, rotated rx 0 ry 90 rz 0 deg; joints [-12.492, -28.278, 112.055, -16.51, -83.169, 50.994]
  Set speed (15.0 mm/s)
  Call Extruder(0.067)
  MoveL 9716 to (496.01, 506.72, 18.3) mm, rotated rx 0 ry 90 rz 0 deg; joints [-12.705, -28.269, 111.994, -16.725, -83.126, 51.031]
  Call Extruder(0.242)
  MoveL 9717 to (504.33, 506.72, 18.3) mm, rotated rx 0 ry 90 rz 0 deg; joints [-12.535, -28.109, 111, -16.585, -82.322, 51.253]
  Call Extruder(0.027)
  MoveL 9718 to (504.33, 505.8, 18.3) mm, rotated rx 0 ry 90 rz 0 deg; joints [-12.452, -28.113, 111.024, -16.5, -82.338, 51.237]
  Call Extruder(0.306)
  MoveL 9719 to (499.53, 496.43, 18.3) mm, rotated rx 0 ry 90 rz 0 deg; joints [-11.69, -28.245, 111.839, -15.708, -82.969, 50.959]
  Call Extruder(0.017)
  MoveL 9720 to (499.27, 495.92, 18.3) mm, rotated rx 0 ry 90 rz 0 deg; joints [-11.648, -28.251, 111.882, -15.665, -83.003, 50.945]
  Call Extruder(0.010)
  MoveL 9721 to (499.84, 495.92, 18.3) mm, rotated rx 0 ry 90 rz 0 deg; joints [-11.637, -28.241, 111.814, -15.656, -82.947, 50.959]
  Call Extruder(0.000)
  MoveL 9722 to (499.84, 495.92, 18.3) mm, rotated rx 0 ry 90 rz 0 deg; joints [-11.637, -28.241, 111.814, -15.656, -82.947, 50.959]
  Call Extruder(0.136)
  MoveL 9723 to (504.51, 495.92, 18.3) mm, rotated rx 0 ry 90 rz 0 deg; joints [-11.55, -28.151, 111.254, -15.584, -82.492, 51.077]
  Call Extruder(0.067)
  MoveL 9724 to (504.51, 493.61, 18.3) mm, rotated rx 0 ry 90 rz 0 deg; joints [-11.338, -28.16, 111.311, -15.369, -82.531, 51.04]
  Call Extruder(0.250)
  MoveL 9725 to (495.92, 493.61, 18.3) mm, rotated rx 0 ry 90 rz 0 deg; joints [-11.498, -28.322, 112.338, -15.501, -83.37, 50.825]
  Call Extruder(0.027)
  MoveL 9726 to (495.92, 494.52, 18.3) mm, rotated rx 0 ry 90 rz 0 deg; joints [-11.583, -28.319, 112.316, -15.587, -83.354, 50.838]
  Call Extruder(0.306)
  MoveL 9727 to (500.7, 503.9, 18.3) mm, rotated rx 0 ry 90 rz 0 deg; joints [-12.351, -28.192, 111.508, -16.384, -82.723, 51.11]
  Call Extruder(0.017)
  MoveL 9728 to (500.96, 504.41, 18.3) mm, rotated rx 0 ry 90 rz 0 deg; joints [-12.392, -28.185, 111.464, -16.427, -82.689, 51.125]
  Call Extruder(0.010)
  MoveL 9729 to (500.39, 504.41, 18.3) mm, rotated rx 0 ry 90 rz 0 deg; joints [-12.404, -28.196, 111.532, -16.436, -82.744, 51.11]
  Call Extruder(0.000)
  MoveL 9730 to (500.39, 504.41, 18.3) mm, rotated rx 0 ry 90 rz 0 deg; joints [-12.404, -28.196, 111.532, -16.436, -82.744, 51.11]
  Call Extruder(0.128)
  MoveL 9731 to (496.01, 504.41, 18.3) mm, rotated rx 0 ry 90 rz 0 deg; joints [-12.492, -28.278, 112.055, -16.51, -83.169, 50.994]
  Set speed (120.0 mm/s)
  MoveL 9732 to (496.01, 504.81, 18.3) mm, rotated rx 0 ry 90 rz 0 deg; joints [-12.529, -28.277, 112.044, -16.547, -83.161, 51]
  Set speed (1000.0 mm/s)
  MoveL 9733 to (495.91, 504.81, 18.3) mm, rotated rx 0 ry 90 rz 0 deg; joints [-12.531, -28.279, 112.056, -16.549, -83.171, 50.997]
  Set speed (1000.0 mm/s)
  MoveL 9734 to (490.47, 509.53, 18.3) mm, rotated rx 0 ry 90 rz 0 deg; joints [-13.08, -28.357, 112.573, -17.086, -83.607, 50.925]
  Set speed (1000.0 mm/s)
  MoveL 9735 to (490.4, 509.6, 18.3) mm, rotated rx 0 ry 90 rz 0 deg; joints [-13.088, -28.358, 112.58, -17.094, -83.613, 50.924]
  Set speed (15.0 mm/s)
  Call Extruder(0.559)
  MoveL 9736 to (490.4, 490.4, 18.3) mm, rotated rx 0 ry 90 rz 0 deg; joints [-11.303, -28.431, 113.07, -15.287, -83.966, 50.639]
  MoveL 9737 to (509.6, 490.4, 18.3) mm, rotated rx 0 ry 90 rz 0 deg; joints [-10.955, -28.071, 110.774, -14.998, -82.086, 51.112]
  MoveL 9738 to (509.6, 509.6, 18.3) mm, rotated rx 0 ry 90 rz 0 deg; joints [-12.688, -27.988, 110.288, -16.763, -81.761, 51.443]
  MoveL 9739 to (490.4, 509.6, 18.3) mm, rotated rx 0 ry 90 rz 0 deg; joints [-13.088, -28.358, 112.58, -17.094, -83.613, 50.924]
  Set speed (120.0 mm/s)
  MoveL 9740 to (490.4, 509.2, 18.3) mm, rotated rx 0 ry 90 rz 0 deg; joints [-13.051, -28.36, 112.591, -17.057, -83.62, 50.918]
  Set speed (1000.0 mm/s)
  MoveL 9741 to (491.1, 508.9, 18.3) mm, rotated rx 0 ry 90 rz 0 deg; joints [-13.008, -28.349, 112.516, -17.016, -83.559, 50.932]
  Set speed (1000.0 mm/s)
  MoveL 9742 to (490.68, 490.68, 18.3) mm, rotated rx 0 ry 90 rz 0 deg; joints [-11.324, -28.425, 113.031, -15.309, -83.934, 50.65]
  Set speed (1000.0 mm/s)
  MoveL 9743 to (490.68, 490.68, 18.4) mm, rotated rx 0 ry 90 rz 0 deg; joints [-11.324, -28.435, 113.036, -15.309, -83.929, 50.652]
  Set speed (30.0 mm/s)
  Call Extruder(0.249)
  MoveL 9744 to (496.74, 496.74, 18.4) mm, rotated rx 0 ry 90 rz 0 deg; joints [-11.772, -28.306, 112.169, -15.782, -83.231, 50.894]
  MoveL 9745 to (496.86, 496.86, 18.4) mm, rotated rx 0 ry 90 rz 0 deg; joints [-11.781, -28.303, 112.152, -15.791, -83.217, 50.899]
  Set speed (120.0 mm/s)
  MoveL 9746 to (495.64, 494.46, 18.4) mm, rotated rx 0 ry 90 rz 0 deg; joints [-11.582, -28.335, 112.356, -15.586, -83.377, 50.832]
  Set speed (30.0 mm/s)
  Call Extruder(0.204)
  MoveL 9747 to (490.68, 499.42, 18.4) mm, rotated rx 0 ry 90 rz 0 deg; joints [-12.139, -28.404, 112.821, -16.134, -83.773, 50.777]
  Set speed (120.0 mm/s)
  MoveL 9748 to (490.68, 500.58, 18.4) mm, rotated rx 0 ry 90 rz 0 deg; joints [-12.247, -28.4, 112.791, -16.243, -83.752, 50.795]
  Set speed (30.0 mm/s)
  Call Extruder(0.208)
  MoveL 9749 to (495.73, 505.63, 18.4) mm, rotated rx 0 ry 90 rz 0 deg; joints [-12.61, -28.289, 112.061, -16.629, -83.168, 51.007]
  Set speed (120.0 mm/s)
  MoveL 9750 to (495.72, 504.27, 18.4) mm, rotated rx 0 ry 90 rz 0 deg; joints [-12.486, -28.295, 112.097, -16.503, -83.193, 50.986]
  Set speed (30.0 mm/s)
  Call Extruder(0.208)
  MoveL 9751 to (490.68, 509.32, 18.4) mm, rotated rx 0 ry 90 rz 0 deg; joints [-13.056, -28.365, 112.559, -17.063, -83.586, 50.929]
  MoveL 9752 to (490.56, 509.44, 18.4) mm, rotated rx 0 ry 90 rz 0 deg; joints [-13.07, -28.367, 112.571, -17.077, -83.595, 50.928]
  Set speed (120.0 mm/s)
  MoveL 9753 to (497.1, 507, 18.4) mm, rotated rx 0 ry 90 rz 0 deg; joints [-12.708, -28.258, 111.861, -16.733, -83.01, 51.066]
  Set speed (30.0 mm/s)
  Call Extruder(0.096)
  MoveL 9754 to (499.42, 509.32, 18.4) mm, rotated rx 0 ry 90 rz 0 deg; joints [-12.872, -28.204, 111.522, -16.908, -82.742, 51.168]
  Set speed (120.0 mm/s)
  MoveL 9755 to (500.58, 509.32, 18.4) mm, rotated rx 0 ry 90 rz 0 deg; joints [-12.847, -28.182, 111.384, -16.888, -82.63, 51.199]
  Set speed (30.0 mm/s)
  Call Extruder(0.096)
  MoveL 9756 to (502.9, 507, 18.4) mm, rotated rx 0 ry 90 rz 0 deg; joints [-12.589, -28.146, 111.169, -16.634, -82.449, 51.221]
  MoveL 9757 to (503.02, 506.87, 18.4) mm, rotated rx 0 ry 90 rz 0 deg; joints [-12.575, -28.145, 111.157, -16.621, -82.439, 51.222]
  Set speed (120.0 mm/s)
  MoveL 9758 to (504.46, 505.44, 18.4) mm, rotated rx 0 ry 90 rz 0 deg; joints [-12.416, -28.122, 111.023, -16.465, -82.327, 51.236]
  Set speed (30.0 mm/s)
  Call Extruder(0.200)
  MoveL 9759 to (509.32, 500.58, 18.4) mm, rotated rx 0 ry 90 rz 0 deg; joints [-11.882, -28.045, 110.564, -15.941, -81.941, 51.277]
  Set speed (120.0 mm/s)
  MoveL 9760 to (509.32, 499.42, 18.4) mm, rotated rx 0 ry 90 rz 0 deg; joints [-11.777, -28.05, 110.594, -15.834, -81.961, 51.257]
  Set speed (30.0 mm/s)
  Call Extruder(0.186)
  MoveL 9761 to (504.79, 494.89, 18.4) mm, rotated rx 0 ry 90 rz 0 deg; joints [-11.45, -28.16, 111.251, -15.484, -82.477, 51.069]
  Set speed (120.0 mm/s)
  MoveL 9762 to (504.79, 495.21, 18.4) mm, rotated rx 0 ry 90 rz 0 deg; joints [-11.479, -28.159, 111.243, -15.514, -82.472, 51.074]
  Set speed (30.0 mm/s)
  Call Extruder(0.186)
  MoveL 9763 to (509.32, 490.68, 18.4) mm, rotated rx 0 ry 90 rz 0 deg; joints [-10.985, -28.086, 110.806, -15.028, -82.104, 51.111]
  MoveL 9764 to (509.44, 490.56, 18.4) mm, rotated rx 0 ry 90 rz 0 deg; joints [-10.972, -28.084, 110.794, -15.015, -82.094, 51.112]
  Set speed (120.0 mm/s)
  MoveL 9765 to (503.23, 493.33, 18.4) mm, rotated rx 0 ry 90 rz 0 deg; joints [-11.336, -28.197, 111.477, -15.363, -82.656, 51.005]
  Set speed (30.0 mm/s)
  Call Extruder(0.109)
  MoveL 9766 to (500.58, 490.68, 18.4) mm, rotated rx 0 ry 90 rz 0 deg; joints [-11.141, -28.257, 111.857, -15.156, -82.958, 50.898]
  Set speed (120.0 mm/s)
  MoveL 9767 to (499.42, 490.68, 18.4) mm, rotated rx 0 ry 90 rz 0 deg; joints [-11.163, -28.279, 111.996, -15.173, -83.072, 50.87]
  Set speed (30.0 mm/s)
  MoveL 9768 to (496.77, 493.33, 18.4) mm, rotated rx 0 ry 90 rz 0 deg; joints [-11.456, -28.318, 112.249, -15.462, -83.286, 50.843]
  MoveL 9769 to (496.65, 493.45, 18.4) mm, rotated rx 0 ry 90 rz 0 deg; joints [-11.47, -28.32, 112.26, -15.475, -83.296, 50.842]
  Set speed (120.0 mm/s)
  MoveL 9770 to (504.54, 493.58, 18.4) mm, rotated rx 0 ry 90 rz 0 deg; joints [-11.335, -28.17, 111.313, -15.366, -82.523, 51.041]
  Set speed (1000.0 mm/s)
  MoveL 9771 to (504.54, 495.95, 18.4) mm, rotated rx 0 ry 90 rz 0 deg; joints [-11.552, -28.161, 111.255, -15.586, -82.484, 51.079]
  Set speed (1000.0 mm/s)
  MoveL 9772 to (501.11, 498.89, 18.4) mm, rotated rx 0 ry 90 rz 0 deg; joints [-11.886, -28.216, 111.594, -15.913, -82.768, 51.04]
  Set speed (30.0 mm/s)
  Call Extruder(0.111)
  MoveL 9773 to (503.8, 496.2, 18.4) mm, rotated rx 0 ry 90 rz 0 deg; joints [-11.588, -28.174, 111.338, -15.621, -82.552, 51.065]
  MoveL 9774 to (503.92, 496.08, 18.4) mm, rotated rx 0 ry 90 rz 0 deg; joints [-11.575, -28.172, 111.327, -15.607, -82.542, 51.066]
  Set speed (120.0 mm/s)
  MoveL 9775 to (504.54, 493.58, 18.4) mm, rotated rx 0 ry 90 rz 0 deg; joints [-11.335, -28.17, 111.313, -15.366, -82.523, 51.041]
  Set speed (1000.0 mm/s)
  MoveL 9776 to (495.89, 493.58, 18.4) mm, rotated rx 0 ry 90 rz 0 deg; joints [-11.496, -28.333, 112.347, -15.499, -83.368, 50.825]
  Set speed (1000.0 mm/s)
  MoveL 9777 to (498.94, 501.06, 18.4) mm, rotated rx 0 ry 90 rz 0 deg; joints [-12.126, -28.248, 111.798, -16.149, -82.94, 51.019]
  Set speed (30.0 mm/s)
  Call Extruder(0.126)
  MoveL 9778 to (495.87, 504.12, 18.4) mm, rotated rx 0 ry 90 rz 0 deg; joints [-12.469, -28.293, 112.083, -16.486, -83.182, 50.987]
  MoveL 9779 to (495.75, 504.25, 18.4) mm, rotated rx 0 ry 90 rz 0 deg; joints [-12.483, -28.294, 112.095, -16.5, -83.191, 50.986]
  Set speed (120.0 mm/s)
  MoveL 9780 to (495.98, 506.75, 18.4) mm, rotated rx 0 ry 90 rz 0 deg; joints [-12.708, -28.28, 112.001, -16.729, -83.123, 51.032]
  Set speed (1000.0 mm/s)
  MoveL 9781 to (504.36, 506.75, 18.4) mm, rotated rx 0 ry 90 rz 0 deg; joints [-12.537, -28.119, 111.001, -16.587, -82.313, 51.255]
  Set speed (1000.0 mm/s)
  MoveL 9782 to (503.43, 503.43, 18.4) mm, rotated rx 0 ry 90 rz 0 deg; joints [-12.254, -28.152, 111.2, -16.296, -82.463, 51.174]
  Set speed (30.0 mm/s)
  Call Extruder(0.243)
  MoveL 9783 to (509.32, 509.32, 18.4) mm, rotated rx 0 ry 90 rz 0 deg; joints [-12.669, -28.006, 110.335, -16.742, -81.788, 51.432]
  MoveL 9784 to (509.44, 509.44, 18.4) mm, rotated rx 0 ry 90 rz 0 deg; joints [-12.677, -28.003, 110.317, -16.752, -81.774, 51.437]
  Set speed (120.0 mm/s)
  MoveL 9785 to (495.98, 506.75, 18.4) mm, rotated rx 0 ry 90 rz 0 deg; joints [-12.708, -28.28, 112.001, -16.729, -83.123, 51.032]
  Set speed (1000.0 mm/s)
  MoveL 9786 to (495.94, 504.34, 18.4) mm, rotated rx 0 ry 90 rz 0 deg; joints [-12.487, -28.291, 112.07, -16.505, -83.172, 50.992]
  Set speed (1000.0 mm/s)
  MoveL 9787 to (496.01, 504.4, 18.4) mm, rotated rx 0 ry 90 rz 0 deg; joints [-12.492, -28.289, 112.06, -16.51, -83.164, 50.995]
  Set speed (15.0 mm/s)
  Call Extruder(0.067)
  MoveL 9788 to (496.01, 506.72, 18.4) mm, rotated rx 0 ry 90 rz 0 deg; joints [-12.705, -28.28, 111.999, -16.726, -83.12, 51.032]
  Call Extruder(0.242)
  MoveL 9789 to (504.33, 506.72, 18.4) mm, rotated rx 0 ry 90 rz 0 deg; joints [-12.535, -28.119, 111.005, -16.585, -82.316, 51.254]
  Call Extruder(0.027)
  MoveL 9790 to (504.33, 505.8, 18.4) mm, rotated rx 0 ry 90 rz 0 deg; joints [-12.452, -28.123, 111.029, -16.501, -82.333, 51.238]
  Call Extruder(0.306)
  MoveL 9791 to (499.53, 496.43, 18.4) mm, rotated rx 0 ry 90 rz 0 deg; joints [-11.69, -28.255, 111.844, -15.708, -82.964, 50.961]
  Call Extruder(0.017)
  MoveL 9792 to (499.27, 495.92, 18.4) mm, rotated rx 0 ry 90 rz 0 deg; joints [-11.648, -28.262, 111.887, -15.665, -82.998, 50.946]
  Call Extruder(0.010)
  MoveL 9793 to (499.84, 495.92, 18.4) mm, rotated rx 0 ry 90 rz 0 deg; joints [-11.637, -28.251, 111.819, -15.656, -82.942, 50.961]
  Call Extruder(0.000)
  MoveL 9794 to (499.84, 495.92, 18.4) mm, rotated rx 0 ry 90 rz 0 deg; joints [-11.637, -28.251, 111.819, -15.656, -82.942, 50.961]
  Call Extruder(0.136)
  MoveL 9795 to (504.51, 495.92, 18.4) mm, rotated rx 0 ry 90 rz 0 deg; joints [-11.55, -28.161, 111.259, -15.584, -82.487, 51.078]
  Call Extruder(0.067)
  MoveL 9796 to (504.51, 493.61, 18.4) mm, rotated rx 0 ry 90 rz 0 deg; joints [-11.338, -28.171, 111.316, -15.369, -82.526, 51.041]
  Call Extruder(0.250)
  MoveL 9797 to (495.92, 493.61, 18.4) mm, rotated rx 0 ry 90 rz 0 deg; joints [-11.498, -28.333, 112.343, -15.502, -83.365, 50.826]
  Call Extruder(0.027)
  MoveL 9798 to (495.92, 494.52, 18.4) mm, rotated rx 0 ry 90 rz 0 deg; joints [-11.583, -28.329, 112.321, -15.587, -83.349, 50.84]
  Call Extruder(0.306)
  MoveL 9799 to (500.7, 503.9, 18.4) mm, rotated rx 0 ry 90 rz 0 deg; joints [-12.351, -28.203, 111.513, -16.384, -82.718, 51.111]
  Call Extruder(0.017)
  MoveL 9800 to (500.96, 504.41, 18.4) mm, rotated rx 0 ry 90 rz 0 deg; joints [-12.392, -28.195, 111.469, -16.427, -82.683, 51.126]
  Call Extruder(0.010)
  MoveL 9801 to (500.39, 504.4, 18.4) mm, rotated rx 0 ry 90 rz 0 deg; joints [-12.404, -28.206, 111.537, -16.436, -82.739, 51.111]
  Call Extruder(0.000)
  MoveL 9802 to (500.39, 504.41, 18.4) mm, rotated rx 0 ry 90 rz 0 deg; joints [-12.404, -28.206, 111.537, -16.436, -82.739, 51.111]
  Call Extruder(0.128)
  MoveL 9803 to (496.01, 504.4, 18.4) mm, rotated rx 0 ry 90 rz 0 deg; joints [-12.492, -28.289, 112.06, -16.51, -83.164, 50.995]
  Set speed (120.0 mm/s)
  MoveL 9804 to (496.01, 504.81, 18.4) mm, rotated rx 0 ry 90 rz 0 deg; joints [-12.529, -28.287, 112.05, -16.547, -83.156, 51.002]
  Set speed (1000.0 mm/s)
  MoveL 9805 to (495.91, 504.81, 18.4) mm, rotated rx 0 ry 90 rz 0 deg; joints [-12.531, -28.289, 112.061, -16.549, -83.166, 50.999]
  Set speed (1000.0 mm/s)
  MoveL 9806 to (490.47, 509.53, 18.4) mm, rotated rx 0 ry 90 rz 0 deg; joints [-13.08, -28.368, 112.578, -17.087, -83.602, 50.927]
  Set speed (1000.0 mm/s)
  MoveL 9807 to (490.4, 509.6, 18.4) mm, rotated rx 0 ry 90 rz 0 deg; joints [-13.088, -28.369, 112.585, -17.094, -83.607, 50.926]
  Set speed (15.0 mm/s)
  Call Extruder(0.559)
  MoveL 9808 to (490.4, 490.4, 18.4) mm, rotated rx 0 ry 90 rz 0 deg; joints [-11.303, -28.441, 113.076, -15.287, -83.961, 50.641]
  MoveL 9809 to (509.6, 490.4, 18.4) mm, rotated rx 0 ry 90 rz 0 deg; joints [-10.955, -28.081, 110.779, -14.998, -82.081, 51.113]
  MoveL 9810 to (509.6, 509.6, 18.4) mm, rotated rx 0 ry 90 rz 0 deg; joints [-12.688, -27.998, 110.293, -16.764, -81.756, 51.444]
  MoveL 9811 to (490.4, 509.6, 18.4) mm, rotated rx 0 ry 90 rz 0 deg; joints [-13.088, -28.369, 112.585, -17.094, -83.607, 50.926]
  Set speed (120.0 mm/s)
  MoveL 9812 to (490.4, 509.2, 18.4) mm, rotated rx 0 ry 90 rz 0 deg; joints [-13.051, -28.371, 112.596, -17.057, -83.615, 50.92]
  Set speed (1000.0 mm/s)
  MoveL 9813 to (491.1, 508.9, 18.4) mm, rotated rx 0 ry 90 rz 0 deg; joints [-13.008, -28.36, 112.521, -17.016, -83.553, 50.934]
  Set speed (1000.0 mm/s)
  MoveL 9814 to (490.68, 490.68, 18.4) mm, rotated rx 0 ry 90 rz 0 deg; joints [-11.324, -28.435, 113.036, -15.309, -83.929, 50.652]
  Set speed (1000.0 mm/s)
  MoveL 9815 to (490.68, 490.68, 18.5) mm, rotated rx 0 ry 90 rz 0 deg; joints [-11.324, -28.446, 113.041, -15.309, -83.923, 50.653]
  Set speed (30.0 mm/s)
  Call Extruder(0.249)
  MoveL 9816 to (496.74, 496.74, 18.5) mm, rotated rx 0 ry 90 rz 0 deg; joints [-11.772, -28.317, 112.174, -15.782, -83.225, 50.896]
  MoveL 9817 to (496.86, 496.86, 18.5) mm, rotated rx 0 ry 90 rz 0 deg; joints [-11.781, -28.314, 112.157, -15.791, -83.211, 50.901]
  Set speed (120.0 mm/s)
  MoveL 9818 to (495.64, 494.46, 18.5) mm, rotated rx 0 ry 90 rz 0 deg; joints [-11.582, -28.345, 112.361, -15.586, -83.372, 50.833]
  Set speed (30.0 mm/s)
  Call Extruder(0.204)
  MoveL 9819 to (490.68, 499.42, 18.5) mm, rotated rx 0 ry 90 rz 0 deg; joints [-12.139, -28.415, 112.826, -16.134, -83.768, 50.779]
  Set speed (120.0 mm/s)
  MoveL 9820 to (490.68, 500.58, 18.5) mm, rotated rx 0 ry 90 rz 0 deg; joints [-12.247, -28.41, 112.796, -16.243, -83.746, 50.796]
  Set speed (30.0 mm/s)
  Call Extruder(0.208)
  MoveL 9821 to (495.73, 505.63, 18.5) mm, rotated rx 0 ry 90 rz 0 deg; joints [-12.61, -28.3, 112.066, -16.629, -83.163, 51.009]
  Set speed (120.0 mm/s)
  MoveL 9822 to (495.73, 504.27, 18.5) mm, rotated rx 0 ry 90 rz 0 deg; joints [-12.486, -28.305, 112.102, -16.503, -83.188, 50.987]
  Set speed (30.0 mm/s)
  Call Extruder(0.208)
  MoveL 9823 to (490.68, 509.32, 18.5) mm, rotated rx 0 ry 90 rz 0 deg; joints [-13.056, -28.376, 112.565, -17.063, -83.58, 50.931]
  MoveL 9824 to (490.56, 509.44, 18.5) mm, rotated rx 0 ry 90 rz 0 deg; joints [-13.07, -28.378, 112.576, -17.077, -83.59, 50.929]
  Set speed (120.0 mm/s)
  MoveL 9825 to (497.1, 507, 18.5) mm, rotated rx 0 ry 90 rz 0 deg; joints [-12.708, -28.269, 111.866, -16.733, -83.004, 51.068]
  Set speed (30.0 mm/s)
  Call Extruder(0.096)
  MoveL 9826 to (499.42, 509.32, 18.5) mm, rotated rx 0 ry 90 rz 0 deg; joints [-12.872, -28.215, 111.527, -16.908, -82.737, 51.169]
  Set speed (120.0 mm/s)
  MoveL 9827 to (500.58, 509.32, 18.5) mm, rotated rx 0 ry 90 rz 0 deg; joints [-12.847, -28.192, 111.389, -16.888, -82.625, 51.2]
  Set speed (30.0 mm/s)
  Call Extruder(0.096)
  MoveL 9828 to (502.9, 507, 18.5) mm, rotated rx 0 ry 90 rz 0 deg; joints [-12.589, -28.157, 111.174, -16.634, -82.444, 51.223]
  MoveL 9829 to (503.02, 506.87, 18.5) mm, rotated rx 0 ry 90 rz 0 deg; joints [-12.575, -28.155, 111.162, -16.621, -82.434, 51.224]
  Set speed (120.0 mm/s)
  MoveL 9830 to (504.46, 505.44, 18.5) mm, rotated rx 0 ry 90 rz 0 deg; joints [-12.416, -28.133, 111.028, -16.465, -82.322, 51.237]
  Set speed (30.0 mm/s)
  Call Extruder(0.200)
  MoveL 9831 to (509.32, 500.58, 18.5) mm, rotated rx 0 ry 90 rz 0 deg; joints [-11.882, -28.056, 110.569, -15.941, -81.936, 51.279]
  Set speed (120.0 mm/s)
  MoveL 9832 to (509.32, 499.42, 18.5) mm, rotated rx 0 ry 90 rz 0 deg; joints [-11.777, -28.061, 110.599, -15.834, -81.956, 51.259]
  Set speed (30.0 mm/s)
  Call Extruder(0.186)
  MoveL 9833 to (504.79, 494.89, 18.5) mm, rotated rx 0 ry 90 rz 0 deg; joints [-11.45, -28.171, 111.256, -15.484, -82.472, 51.07]
  Set speed (120.0 mm/s)
  MoveL 9834 to (504.79, 495.21, 18.5) mm, rotated rx 0 ry 90 rz 0 deg; joints [-11.479, -28.169, 111.248, -15.514, -82.467, 51.075]
  Set speed (30.0 mm/s)
  Call Extruder(0.186)
  MoveL 9835 to (509.32, 490.68, 18.5) mm, rotated rx 0 ry 90 rz 0 deg; joints [-10.985, -28.097, 110.811, -15.028, -82.099, 51.113]
  MoveL 9836 to (509.44, 490.56, 18.5) mm, rotated rx 0 ry 90 rz 0 deg; joints [-10.972, -28.095, 110.799, -15.015, -82.089, 51.114]
  Set speed (120.0 mm/s)
  MoveL 9837 to (503.23, 493.33, 18.5) mm, rotated rx 0 ry 90 rz 0 deg; joints [-11.336, -28.207, 111.482, -15.363, -82.65, 51.006]
  Set speed (30.0 mm/s)
  Call Extruder(0.109)
  MoveL 9838 to (500.58, 490.68, 18.5) mm, rotated rx 0 ry 90 rz 0 deg; joints [-11.141, -28.268, 111.862, -15.156, -82.953, 50.9]
  Set speed (120.0 mm/s)
  MoveL 9839 to (499.42, 490.68, 18.5) mm, rotated rx 0 ry 90 rz 0 deg; joints [-11.163, -28.29, 112.001, -15.173, -83.066, 50.871]
  Set speed (30.0 mm/s)
  MoveL 9840 to (496.77, 493.33, 18.5) mm, rotated rx 0 ry 90 rz 0 deg; joints [-11.456, -28.329, 112.254, -15.462, -83.281, 50.845]
  MoveL 9841 to (496.65, 493.45, 18.5) mm, rotated rx 0 ry 90 rz 0 deg; joints [-11.47, -28.331, 112.265, -15.476, -83.291, 50.844]
  Set speed (120.0 mm/s)
  MoveL 9842 to (504.54, 493.58, 18.5) mm, rotated rx 0 ry 90 rz 0 deg; joints [-11.335, -28.181, 111.318, -15.367, -82.518, 51.043]
  Set speed (1000.0 mm/s)
  MoveL 9843 to (504.54, 495.95, 18.5) mm, rotated rx 0 ry 90 rz 0 deg; joints [-11.552, -28.171, 111.26, -15.586, -82.479, 51.081]
  Set speed (1000.0 mm/s)
  MoveL 9844 to (501.11, 498.89, 18.5) mm, rotated rx 0 ry 90 rz 0 deg; joints [-11.886, -28.226, 111.599, -15.913, -82.762, 51.041]
  Set speed (30.0 mm/s)
  Call Extruder(0.111)
  MoveL 9845 to (503.8, 496.2, 18.5) mm, rotated rx 0 ry 90 rz 0 deg; joints [-11.588, -28.185, 111.343, -15.621, -82.547, 51.066]
  MoveL 9846 to (503.92, 496.08, 18.5) mm, rotated rx 0 ry 90 rz 0 deg; joints [-11.575, -28.183, 111.332, -15.608, -82.537, 51.067]
  Set speed (120.0 mm/s)
  MoveL 9847 to (504.54, 493.58, 18.5) mm, rotated rx 0 ry 90 rz 0 deg; joints [-11.335, -28.181, 111.318, -15.367, -82.518, 51.043]
  Set speed (1000.0 mm/s)
  MoveL 9848 to (495.89, 493.58, 18.5) mm, rotated rx 0 ry 90 rz 0 deg; joints [-11.496, -28.344, 112.352, -15.5, -83.362, 50.827]
  Set speed (1000.0 mm/s)
  MoveL 9849 to (498.94, 501.06, 18.5) mm, rotated rx 0 ry 90 rz 0 deg; joints [-12.126, -28.259, 111.803, -16.149, -82.934, 51.02]
  Set speed (30.0 mm/s)
  Call Extruder(0.126)
  MoveL 9850 to (495.87, 504.12, 18.5) mm, rotated rx 0 ry 90 rz 0 deg; joints [-12.469, -28.303, 112.088, -16.486, -83.176, 50.989]
  MoveL 9851 to (495.75, 504.25, 18.5) mm, rotated rx 0 ry 90 rz 0 deg; joints [-12.483, -28.305, 112.1, -16.5, -83.186, 50.987]
  Set speed (120.0 mm/s)
  MoveL 9852 to (495.98, 506.75, 18.5) mm, rotated rx 0 ry 90 rz 0 deg; joints [-12.708, -28.291, 112.006, -16.729, -83.117, 51.034]
  Set speed (1000.0 mm/s)
  MoveL 9853 to (504.35, 506.75, 18.5) mm, rotated rx 0 ry 90 rz 0 deg; joints [-12.537, -28.129, 111.006, -16.587, -82.308, 51.257]
  Set speed (1000.0 mm/s)
  MoveL 9854 to (503.43, 503.43, 18.5) mm, rotated rx 0 ry 90 rz 0 deg; joints [-12.254, -28.162, 111.205, -16.296, -82.457, 51.176]
  Set speed (30.0 mm/s)
  Call Extruder(0.243)
  MoveL 9855 to (509.32, 509.32, 18.5) mm, rotated rx 0 ry 90 rz 0 deg; joints [-12.669, -28.016, 110.34, -16.743, -81.783, 51.433]
  MoveL 9856 to (509.44, 509.44, 18.5) mm, rotated rx 0 ry 90 rz 0 deg; joints [-12.677, -28.013, 110.322, -16.752, -81.769, 51.439]
  Set speed (120.0 mm/s)
  MoveL 9857 to (495.98, 506.75, 18.5) mm, rotated rx 0 ry 90 rz 0 deg; joints [-12.708, -28.291, 112.006, -16.729, -83.117, 51.034]
  Set speed (1000.0 mm/s)
  MoveL 9858 to (495.94, 504.33, 18.5) mm, rotated rx 0 ry 90 rz 0 deg; joints [-12.487, -28.301, 112.075, -16.505, -83.166, 50.994]
  Set speed (1000.0 mm/s)
  MoveL 9859 to (496.01, 504.4, 18.5) mm, rotated rx 0 ry 90 rz 0 deg; joints [-12.492, -28.3, 112.065, -16.51, -83.158, 50.997]
  Set speed (15.0 mm/s)
  Call Extruder(0.067)
  MoveL 9860 to (496.01, 506.72, 18.5) mm, rotated rx 0 ry 90 rz 0 deg; joints [-12.705, -28.29, 112.004, -16.726, -83.115, 51.034]
  Call Extruder(0.242)
  MoveL 9861 to (504.33, 506.72, 18.5) mm, rotated rx 0 ry 90 rz 0 deg; joints [-12.535, -28.13, 111.01, -16.585, -82.311, 51.256]
  Call Extruder(0.027)
  MoveL 9862 to (504.33, 505.8, 18.5) mm, rotated rx 0 ry 90 rz 0 deg; joints [-12.452, -28.134, 111.034, -16.501, -82.328, 51.24]
  Call Extruder(0.306)
  MoveL 9863 to (499.53, 496.43, 18.5) mm, rotated rx 0 ry 90 rz 0 deg; joints [-11.69, -28.266, 111.849, -15.709, -82.958, 50.962]
  Call Extruder(0.017)
  MoveL 9864 to (499.27, 495.92, 18.5) mm, rotated rx 0 ry 90 rz 0 deg; joints [-11.648, -28.273, 111.892, -15.665, -82.992, 50.948]
  Call Extruder(0.010)
  MoveL 9865 to (499.84, 495.92, 18.5) mm, rotated rx 0 ry 90 rz 0 deg; joints [-11.637, -28.262, 111.824, -15.656, -82.937, 50.962]
  Call Extruder(0.000)
  MoveL 9866 to (499.84, 495.92, 18.5) mm, rotated rx 0 ry 90 rz 0 deg; joints [-11.637, -28.262, 111.824, -15.656, -82.937, 50.962]
  Call Extruder(0.136)
  MoveL 9867 to (504.51, 495.92, 18.5) mm, rotated rx 0 ry 90 rz 0 deg; joints [-11.55, -28.172, 111.264, -15.584, -82.482, 51.08]
  Call Extruder(0.067)
  MoveL 9868 to (504.51, 493.61, 18.5) mm, rotated rx 0 ry 90 rz 0 deg; joints [-11.338, -28.181, 111.321, -15.37, -82.52, 51.042]
  Call Extruder(0.250)
  MoveL 9869 to (495.92, 493.61, 18.5) mm, rotated rx 0 ry 90 rz 0 deg; joints [-11.498, -28.343, 112.348, -15.502, -83.359, 50.828]
  Call Extruder(0.027)
  MoveL 9870 to (495.92, 494.52, 18.5) mm, rotated rx 0 ry 90 rz 0 deg; joints [-11.583, -28.34, 112.326, -15.588, -83.343, 50.841]
  Call Extruder(0.306)
  MoveL 9871 to (500.7, 503.9, 18.5) mm, rotated rx 0 ry 90 rz 0 deg; joints [-12.351, -28.213, 111.518, -16.384, -82.712, 51.113]
  Call Extruder(0.017)
  MoveL 9872 to (500.96, 504.4, 18.5) mm, rotated rx 0 ry 90 rz 0 deg; joints [-12.392, -28.206, 111.474, -16.427, -82.678, 51.128]
  Call Extruder(0.010)
  MoveL 9873 to (500.39, 504.41, 18.5) mm, rotated rx 0 ry 90 rz 0 deg; joints [-12.404, -28.217, 111.542, -16.436, -82.733, 51.113]
  Call Extruder(0.000)
  MoveL 9874 to (500.39, 504.41, 18.5) mm, rotated rx 0 ry 90 rz 0 deg; joints [-12.404, -28.217, 111.542, -16.436, -82.733, 51.113]
  Call Extruder(0.128)
  MoveL 9875 to (496.01, 504.4, 18.5) mm, rotated rx 0 ry 90 rz 0 deg; joints [-12.492, -28.3, 112.065, -16.51, -83.158, 50.997]
  Set speed (120.0 mm/s)
  MoveL 9876 to (496.01, 504.81, 18.5) mm, rotated rx 0 ry 90 rz 0 deg; joints [-12.529, -28.298, 112.055, -16.548, -83.151, 51.003]
  Set speed (1000.0 mm/s)
  MoveL 9877 to (495.91, 504.81, 18.5) mm, rotated rx 0 ry 90 rz 0 deg; joints [-12.531, -28.3, 112.067, -16.549, -83.161, 51]
  Set speed (1000.0 mm/s)
  MoveL 9878 to (490.47, 509.53, 18.5) mm, rotated rx 0 ry 90 rz 0 deg; joints [-13.08, -28.379, 112.583, -17.087, -83.596, 50.928]
  Set speed (1000.0 mm/s)
  MoveL 9879 to (490.4, 509.6, 18.5) mm, rotated rx 0 ry 90 rz 0 deg; joints [-13.088, -28.38, 112.59, -17.095, -83.602, 50.928]
  Set speed (15.0 mm/s)
  Call Extruder(0.559)
  MoveL 9880 to (490.4, 490.4, 18.5) mm, rotated rx 0 ry 90 rz 0 deg; joints [-11.303, -28.452, 113.081, -15.287, -83.956, 50.642]
  MoveL 9881 to (509.6, 490.4, 18.5) mm, rotated rx 0 ry 90 rz 0 deg; joints [-10.955, -28.092, 110.784, -14.999, -82.076, 51.115]
  MoveL 9882 to (509.6, 509.6, 18.5) mm, rotated rx 0 ry 90 rz 0 deg; joints [-12.688, -28.009, 110.298, -16.764, -81.751, 51.446]
  MoveL 9883 to (490.4, 509.6, 18.5) mm, rotated rx 0 ry 90 rz 0 deg; joints [-13.088, -28.38, 112.59, -17.095, -83.602, 50.928]
  Set speed (120.0 mm/s)
  MoveL 9884 to (490.4, 509.2, 18.5) mm, rotated rx 0 ry 90 rz 0 deg; joints [-13.051, -28.381, 112.601, -17.057, -83.61, 50.921]
  Set speed (1000.0 mm/s)
  MoveL 9885 to (491.1, 508.9, 18.5) mm, rotated rx 0 ry 90 rz 0 deg; joints [-13.008, -28.37, 112.526, -17.016, -83.548, 50.936]
  Set speed (1000.0 mm/s)
  MoveL 9886 to (490.68, 490.68, 18.5) mm, rotated rx 0 ry 90 rz 0 deg; joints [-11.324, -28.446, 113.041, -15.309, -83.923, 50.653]
  Set speed (1000.0 mm/s)
  MoveL 9887 to (490.68, 490.68, 18.6) mm, rotated rx 0 ry 90 rz 0 deg; joints [-11.324, -28.457, 113.046, -15.309, -83.918, 50.655]
  Set speed (30.0 mm/s)
  Call Extruder(0.249)
  MoveL 9888 to (496.74, 496.74, 18.6) mm, rotated rx 0 ry 90 rz 0 deg; joints [-11.772, -28.327, 112.18, -15.782, -83.22, 50.897]
  MoveL 9889 to (496.86, 496.86, 18.6) mm, rotated rx 0 ry 90 rz 0 deg; joints [-11.781, -28.324, 112.162, -15.792, -83.206, 50.902]
  Set speed (120.0 mm/s)
  MoveL 9890 to (495.64, 494.46, 18.6) mm, rotated rx 0 ry 90 rz 0 deg; joints [-11.582, -28.356, 112.366, -15.586, -83.367, 50.835]
  Set speed (30.0 mm/s)
  Call Extruder(0.204)
  MoveL 9891 to (490.68, 499.42, 18.6) mm, rotated rx 0 ry 90 rz 0 deg; joints [-12.139, -28.425, 112.831, -16.134, -83.762, 50.78]
  Set speed (120.0 mm/s)
  MoveL 9892 to (490.68, 500.58, 18.6) mm, rotated rx 0 ry 90 rz 0 deg; joints [-12.247, -28.421, 112.802, -16.243, -83.741, 50.798]
  Set speed (30.0 mm/s)
  Call Extruder(0.208)
  MoveL 9893 to (495.73, 505.62, 18.6) mm, rotated rx 0 ry 90 rz 0 deg; joints [-12.61, -28.31, 112.071, -16.629, -83.157, 51.01]
  Set speed (120.0 mm/s)
  MoveL 9894 to (495.73, 504.27, 18.6) mm, rotated rx 0 ry 90 rz 0 deg; joints [-12.486, -28.316, 112.107, -16.503, -83.183, 50.989]
  Set speed (30.0 mm/s)
  Call Extruder(0.208)
  MoveL 9895 to (490.68, 509.32, 18.6) mm, rotated rx 0 ry 90 rz 0 deg; joints [-13.056, -28.387, 112.57, -17.063, -83.575, 50.932]
  MoveL 9896 to (490.56, 509.44, 18.6) mm, rotated rx 0 ry 90 rz 0 deg; joints [-13.07, -28.388, 112.581, -17.077, -83.585, 50.931]
  Set speed (120.0 mm/s)
  MoveL 9897 to (497.1, 507, 18.6) mm, rotated rx 0 ry 90 rz 0 deg; joints [-12.708, -28.279, 111.872, -16.733, -82.999, 51.07]
  Set speed (30.0 mm/s)
  Call Extruder(0.096)
  MoveL 9898 to (499.42, 509.32, 18.6) mm, rotated rx 0 ry 90 rz 0 deg; joints [-12.872, -28.225, 111.532, -16.908, -82.731, 51.171]
  Set speed (120.0 mm/s)
  MoveL 9899 to (500.58, 509.32, 18.6) mm, rotated rx 0 ry 90 rz 0 deg; joints [-12.847, -28.203, 111.394, -16.889, -82.62, 51.202]
  Set speed (30.0 mm/s)
  Call Extruder(0.096)
  MoveL 9900 to (502.9, 507, 18.6) mm, rotated rx 0 ry 90 rz 0 deg; joints [-12.589, -28.167, 111.179, -16.635, -82.438, 51.224]
  MoveL 9901 to (503.02, 506.87, 18.6) mm, rotated rx 0 ry 90 rz 0 deg; joints [-12.575, -28.166, 111.167, -16.621, -82.429, 51.225]
  Set speed (120.0 mm/s)
  MoveL 9902 to (504.46, 505.44, 18.6) mm, rotated rx 0 ry 90 rz 0 deg; joints [-12.416, -28.143, 111.034, -16.465, -82.316, 51.239]
  Set speed (30.0 mm/s)
  Call Extruder(0.200)
  MoveL 9903 to (509.32, 500.58, 18.6) mm, rotated rx 0 ry 90 rz 0 deg; joints [-11.882, -28.066, 110.574, -15.941, -81.931, 51.28]
  Set speed (120.0 mm/s)
  MoveL 9904 to (509.32, 499.42, 18.6) mm, rotated rx 0 ry 90 rz 0 deg; joints [-11.777, -28.071, 110.604, -15.834, -81.95, 51.26]
  Set speed (30.0 mm/s)
  Call Extruder(0.186)
  MoveL 9905 to (504.79, 494.89, 18.6) mm, rotated rx 0 ry 90 rz 0 deg; joints [-11.45, -28.181, 111.261, -15.485, -82.467, 51.071]
  Set speed (120.0 mm/s)
  MoveL 9906 to (504.79, 495.21, 18.6) mm, rotated rx 0 ry 90 rz 0 deg; joints [-11.479, -28.18, 111.253, -15.514, -82.461, 51.077]
  Set speed (30.0 mm/s)
  Call Extruder(0.186)
  MoveL 9907 to (509.32, 490.68, 18.6) mm, rotated rx 0 ry 90 rz 0 deg; joints [-10.985, -28.107, 110.816, -15.029, -82.093, 51.114]
  MoveL 9908 to (509.44, 490.56, 18.6) mm, rotated rx 0 ry 90 rz 0 deg; joints [-10.972, -28.105, 110.804, -15.016, -82.083, 51.115]
  Set speed (120.0 mm/s)
  MoveL 9909 to (503.23, 493.33, 18.6) mm, rotated rx 0 ry 90 rz 0 deg; joints [-11.336, -28.218, 111.487, -15.363, -82.645, 51.008]
  Set speed (30.0 mm/s)
  Call Extruder(0.109)
  MoveL 9910 to (500.58, 490.68, 18.6) mm, rotated rx 0 ry 90 rz 0 deg; joints [-11.141, -28.278, 111.867, -15.156, -82.948, 50.901]
  Set speed (120.0 mm/s)
  MoveL 9911 to (499.42, 490.68, 18.6) mm, rotated rx 0 ry 90 rz 0 deg; joints [-11.163, -28.3, 112.006, -15.174, -83.061, 50.873]
  Set speed (30.0 mm/s)
  MoveL 9912 to (496.77, 493.33, 18.6) mm, rotated rx 0 ry 90 rz 0 deg; joints [-11.456, -28.339, 112.259, -15.462, -83.276, 50.846]
  MoveL 9913 to (496.65, 493.45, 18.6) mm, rotated rx 0 ry 90 rz 0 deg; joints [-11.47, -28.341, 112.27, -15.476, -83.285, 50.845]
  Set speed (120.0 mm/s)
  MoveL 9914 to (504.54, 493.58, 18.6) mm, rotated rx 0 ry 90 rz 0 deg; joints [-11.335, -28.191, 111.323, -15.367, -82.513, 51.044]
  Set speed (1000.0 mm/s)
  MoveL 9915 to (504.54, 495.95, 18.6) mm, rotated rx 0 ry 90 rz 0 deg; joints [-11.552, -28.182, 111.265, -15.586, -82.473, 51.082]
  Set speed (1000.0 mm/s)
  MoveL 9916 to (501.11, 498.89, 18.6) mm, rotated rx 0 ry 90 rz 0 deg; joints [-11.886, -28.237, 111.604, -15.913, -82.757, 51.043]
  Set speed (30.0 mm/s)
  Call Extruder(0.111)
  MoveL 9917 to (503.8, 496.2, 18.6) mm, rotated rx 0 ry 90 rz 0 deg; joints [-11.588, -28.195, 111.348, -15.621, -82.541, 51.068]
  MoveL 9918 to (503.92, 496.08, 18.6) mm, rotated rx 0 ry 90 rz 0 deg; joints [-11.575, -28.193, 111.337, -15.608, -82.531, 51.069]
  Set speed (120.0 mm/s)
  MoveL 9919 to (504.54, 493.58, 18.6) mm, rotated rx 0 ry 90 rz 0 deg; joints [-11.335, -28.191, 111.323, -15.367, -82.513, 51.044]
  Set speed (1000.0 mm/s)
  MoveL 9920 to (495.89, 493.58, 18.6) mm, rotated rx 0 ry 90 rz 0 deg; joints [-11.496, -28.354, 112.357, -15.5, -83.357, 50.828]
  Set speed (1000.0 mm/s)
  MoveL 9921 to (498.94, 501.06, 18.6) mm, rotated rx 0 ry 90 rz 0 deg; joints [-12.126, -28.269, 111.808, -16.15, -82.929, 51.022]
  Set speed (30.0 mm/s)
  Call Extruder(0.126)
  MoveL 9922 to (495.87, 504.12, 18.6) mm, rotated rx 0 ry 90 rz 0 deg; joints [-12.469, -28.314, 112.093, -16.486, -83.171, 50.99]
  MoveL 9923 to (495.75, 504.25, 18.6) mm, rotated rx 0 ry 90 rz 0 deg; joints [-12.483, -28.316, 112.105, -16.5, -83.181, 50.989]
  Set speed (120.0 mm/s)
  MoveL 9924 to (495.98, 506.75, 18.6) mm, rotated rx 0 ry 90 rz 0 deg; joints [-12.708, -28.301, 112.011, -16.729, -83.112, 51.035]
  Set speed (1000.0 mm/s)
  MoveL 9925 to (504.36, 506.75, 18.6) mm, rotated rx 0 ry 90 rz 0 deg; joints [-12.537, -28.14, 111.011, -16.588, -82.303, 51.258]
  Set speed (1000.0 mm/s)
  MoveL 9926 to (503.43, 503.43, 18.6) mm, rotated rx 0 ry 90 rz 0 deg; joints [-12.254, -28.173, 111.21, -16.296, -82.452, 51.178]
  Set speed (30.0 mm/s)
  Call Extruder(0.243)
  MoveL 9927 to (509.32, 509.32, 18.6) mm, rotated rx 0 ry 90 rz 0 deg; joints [-12.669, -28.027, 110.345, -16.743, -81.778, 51.435]
  MoveL 9928 to (509.44, 509.44, 18.6) mm, rotated rx 0 ry 90 rz 0 deg; joints [-12.677, -28.023, 110.327, -16.752, -81.764, 51.441]
  Set speed (120.0 mm/s)
  MoveL 9929 to (495.98, 506.75, 18.6) mm, rotated rx 0 ry 90 rz 0 deg; joints [-12.708, -28.301, 112.011, -16.729, -83.112, 51.035]
  Set speed (1000.0 mm/s)
  MoveL 9930 to (495.94, 504.34, 18.6) mm, rotated rx 0 ry 90 rz 0 deg; joints [-12.487, -28.312, 112.08, -16.505, -83.161, 50.995]
  Set speed (1000.0 mm/s)
  MoveL 9931 to (496.01, 504.41, 18.6) mm, rotated rx 0 ry 90 rz 0 deg; joints [-12.492, -28.31, 112.07, -16.51, -83.153, 50.998]
  Set speed (15.0 mm/s)
  Call Extruder(0.067)
  MoveL 9932 to (496.01, 506.72, 18.6) mm, rotated rx 0 ry 90 rz 0 deg; joints [-12.705, -28.301, 112.009, -16.726, -83.11, 51.036]
  Call Extruder(0.242)
  MoveL 9933 to (504.33, 506.72, 18.6) mm, rotated rx 0 ry 90 rz 0 deg; joints [-12.535, -28.14, 111.015, -16.585, -82.306, 51.257]
  Call Extruder(0.027)
  MoveL 9934 to (504.33, 505.8, 18.6) mm, rotated rx 0 ry 90 rz 0 deg; joints [-12.452, -28.144, 111.04, -16.501, -82.322, 51.241]
  Call Extruder(0.306)
  MoveL 9935 to (499.53, 496.43, 18.6) mm, rotated rx 0 ry 90 rz 0 deg; joints [-11.69, -28.276, 111.854, -15.709, -82.953, 50.964]
  Call Extruder(0.017)
  MoveL 9936 to (499.27, 495.92, 18.6) mm, rotated rx 0 ry 90 rz 0 deg; joints [-11.648, -28.283, 111.897, -15.665, -82.987, 50.949]
  Call Extruder(0.010)
  MoveL 9937 to (499.84, 495.92, 18.6) mm, rotated rx 0 ry 90 rz 0 deg; joints [-11.637, -28.272, 111.829, -15.656, -82.932, 50.964]
  Call Extruder(0.000)
  MoveL 9938 to (499.84, 495.92, 18.6) mm, rotated rx 0 ry 90 rz 0 deg; joints [-11.637, -28.272, 111.829, -15.656, -82.931, 50.964]
  Call Extruder(0.136)
  MoveL 9939 to (504.51, 495.92, 18.6) mm, rotated rx 0 ry 90 rz 0 deg; joints [-11.55, -28.182, 111.269, -15.584, -82.476, 51.081]
  Call Extruder(0.067)
  MoveL 9940 to (504.51, 493.61, 18.6) mm, rotated rx 0 ry 90 rz 0 deg; joints [-11.338, -28.192, 111.326, -15.37, -82.515, 51.044]
  Call Extruder(0.250)
  MoveL 9941 to (495.92, 493.61, 18.6) mm, rotated rx 0 ry 90 rz 0 deg; joints [-11.498, -28.354, 112.353, -15.502, -83.354, 50.829]
  Call Extruder(0.027)
  MoveL 9942 to (495.92, 494.52, 18.6) mm, rotated rx 0 ry 90 rz 0 deg; joints [-11.583, -28.35, 112.331, -15.588, -83.338, 50.843]
  Call Extruder(0.306)
  MoveL 9943 to (500.7, 503.9, 18.6) mm, rotated rx 0 ry 90 rz 0 deg; joints [-12.351, -28.224, 111.523, -16.384, -82.707, 51.114]
  Call Extruder(0.017)
  MoveL 9944 to (500.96, 504.41, 18.6) mm, rotated rx 0 ry 90 rz 0 deg; joints [-12.392, -28.217, 111.479, -16.427, -82.673, 51.129]
  Call Extruder(0.010)
  MoveL 9945 to (500.39, 504.41, 18.6) mm, rotated rx 0 ry 90 rz 0 deg; joints [-12.404, -28.228, 111.547, -16.437, -82.728, 51.114]
  Call Extruder(0.000)
  MoveL 9946 to (500.39, 504.41, 18.6) mm, rotated rx 0 ry 90 rz 0 deg; joints [-12.404, -28.228, 111.547, -16.437, -82.728, 51.114]
  Call Extruder(0.128)
  MoveL 9947 to (496.01, 504.41, 18.6) mm, rotated rx 0 ry 90 rz 0 deg; joints [-12.492, -28.31, 112.07, -16.51, -83.153, 50.998]
  Set speed (120.0 mm/s)
  MoveL 9948 to (496.01, 504.81, 18.6) mm, rotated rx 0 ry 90 rz 0 deg; joints [-12.529, -28.309, 112.06, -16.548, -83.146, 51.005]
  Set speed (1000.0 mm/s)
  MoveL 9949 to (495.91, 504.81, 18.6) mm, rotated rx 0 ry 90 rz 0 deg; joints [-12.531, -28.31, 112.072, -16.549, -83.155, 51.002]
  Set speed (1000.0 mm/s)
  MoveL 9950 to (490.47, 509.53, 18.6) mm, rotated rx 0 ry 90 rz 0 deg; joints [-13.08, -28.389, 112.589, -17.087, -83.591, 50.93]
  Set speed (1000.0 mm/s)
  MoveL 9951 to (490.4, 509.6, 18.6) mm, rotated rx 0 ry 90 rz 0 deg; joints [-13.088, -28.39, 112.595, -17.095, -83.597, 50.929]
  Set speed (15.0 mm/s)
  Call Extruder(0.559)
  MoveL 9952 to (490.4, 490.4, 18.6) mm, rotated rx 0 ry 90 rz 0 deg; joints [-11.303, -28.463, 113.086, -15.287, -83.95, 50.644]
  MoveL 9953 to (509.6, 490.4, 18.6) mm, rotated rx 0 ry 90 rz 0 deg; joints [-10.955, -28.102, 110.789, -14.999, -82.07, 51.116]
  MoveL 9954 to (509.6, 509.6, 18.6) mm, rotated rx 0 ry 90 rz 0 deg; joints [-12.688, -28.019, 110.303, -16.764, -81.746, 51.448]
  MoveL 9955 to (490.4, 509.6, 18.6) mm, rotated rx 0 ry 90 rz 0 deg; joints [-13.088, -28.39, 112.595, -17.095, -83.597, 50.929]
  Set speed (120.0 mm/s)
  MoveL 9956 to (490.4, 509.2, 18.6) mm, rotated rx 0 ry 90 rz 0 deg; joints [-13.051, -28.392, 112.606, -17.057, -83.604, 50.923]
  Set speed (1000.0 mm/s)
  MoveL 9957 to (491.1, 508.9, 18.6) mm, rotated rx 0 ry 90 rz 0 deg; joints [-13.008, -28.381, 112.531, -17.017, -83.543, 50.937]
  Set speed (1000.0 mm/s)
  MoveL 9958 to (490.68, 490.68, 18.6) mm, rotated rx 0 ry 90 rz 0 deg; joints [-11.324, -28.457, 113.046, -15.309, -83.918, 50.655]
  Set speed (1000.0 mm/s)
  MoveL 9959 to (490.68, 490.68, 18.7) mm, rotated rx 0 ry 90 rz 0 deg; joints [-11.324, -28.468, 113.051, -15.31, -83.913, 50.656]
  Set speed (30.0 mm/s)
  Call Extruder(0.249)
  MoveL 9960 to (496.74, 496.74, 18.7) mm, rotated rx 0 ry 90 rz 0 deg; joints [-11.772, -28.338, 112.185, -15.782, -83.215, 50.899]
  MoveL 9961 to (496.86, 496.86, 18.7) mm, rotated rx 0 ry 90 rz 0 deg; joints [-11.781, -28.335, 112.167, -15.792, -83.201, 50.904]
  Set speed (120.0 mm/s)
  MoveL 9962 to (495.64, 494.46, 18.7) mm, rotated rx 0 ry 90 rz 0 deg; joints [-11.582, -28.366, 112.371, -15.586, -83.361, 50.836]
  Set speed (30.0 mm/s)
  Call Extruder(0.204)
  MoveL 9963 to (490.68, 499.42, 18.7) mm, rotated rx 0 ry 90 rz 0 deg; joints [-12.139, -28.436, 112.836, -16.134, -83.757, 50.782]
  Set speed (120.0 mm/s)
  MoveL 9964 to (490.68, 500.58, 18.7) mm, rotated rx 0 ry 90 rz 0 deg; joints [-12.247, -28.432, 112.807, -16.243, -83.736, 50.799]
  Set speed (30.0 mm/s)
  Call Extruder(0.208)
  MoveL 9965 to (495.73, 505.62, 18.7) mm, rotated rx 0 ry 90 rz 0 deg; joints [-12.61, -28.321, 112.076, -16.629, -83.152, 51.012]
  Set speed (120.0 mm/s)
  MoveL 9966 to (495.72, 504.27, 18.7) mm, rotated rx 0 ry 90 rz 0 deg; joints [-12.486, -28.327, 112.112, -16.503, -83.177, 50.99]
  Set speed (30.0 mm/s)
  Call Extruder(0.208)
  MoveL 9967 to (490.68, 509.32, 18.7) mm, rotated rx 0 ry 90 rz 0 deg; joints [-13.056, -28.397, 112.575, -17.064, -83.57, 50.934]
  MoveL 9968 to (490.56, 509.44, 18.7) mm, rotated rx 0 ry 90 rz 0 deg; joints [-13.07, -28.399, 112.586, -17.077, -83.579, 50.933]
  Set speed (120.0 mm/s)
  MoveL 9969 to (497.1, 507, 18.7) mm, rotated rx 0 ry 90 rz 0 deg; joints [-12.708, -28.29, 111.877, -16.733, -82.994, 51.071]
  Set speed (30.0 mm/s)
  Call Extruder(0.096)
  MoveL 9970 to (499.42, 509.32, 18.7) mm, rotated rx 0 ry 90 rz 0 deg; joints [-12.872, -28.236, 111.537, -16.909, -82.726, 51.172]
  Set speed (120.0 mm/s)
  MoveL 9971 to (500.58, 509.32, 18.7) mm, rotated rx 0 ry 90 rz 0 deg; joints [-12.847, -28.213, 111.399, -16.889, -82.614, 51.204]
  Set speed (30.0 mm/s)
  Call Extruder(0.096)
  MoveL 9972 to (502.9, 507, 18.7) mm, rotated rx 0 ry 90 rz 0 deg; joints [-12.589, -28.178, 111.184, -16.635, -82.433, 51.226]
  MoveL 9973 to (503.02, 506.87, 18.7) mm, rotated rx 0 ry 90 rz 0 deg; joints [-12.575, -28.176, 111.172, -16.621, -82.424, 51.227]
  Set speed (120.0 mm/s)
  MoveL 9974 to (504.46, 505.44, 18.7) mm, rotated rx 0 ry 90 rz 0 deg; joints [-12.416, -28.154, 111.039, -16.466, -82.311, 51.24]
  Set speed (30.0 mm/s)
  Call Extruder(0.200)
  MoveL 9975 to (509.32, 500.58, 18.7) mm, rotated rx 0 ry 90 rz 0 deg; joints [-11.882, -28.077, 110.579, -15.941, -81.926, 51.282]
  Set speed (120.0 mm/s)
  MoveL 9976 to (509.32, 499.42, 18.7) mm, rotated rx 0 ry 90 rz 0 deg; joints [-11.777, -28.082, 110.609, -15.835, -81.945, 51.262]
  Set speed (30.0 mm/s)
  Call Extruder(0.186)
  MoveL 9977 to (504.79, 494.89, 18.7) mm, rotated rx 0 ry 90 rz 0 deg; joints [-11.45, -28.192, 111.266, -15.485, -82.461, 51.073]
  Set speed (120.0 mm/s)
  MoveL 9978 to (504.79, 495.21, 18.7) mm, rotated rx 0 ry 90 rz 0 deg; joints [-11.479, -28.19, 111.258, -15.514, -82.456, 51.078]
  Set speed (30.0 mm/s)
  Call Extruder(0.186)
  MoveL 9979 to (509.32, 490.68, 18.7) mm, rotated rx 0 ry 90 rz 0 deg; joints [-10.985, -28.118, 110.821, -15.029, -82.088, 51.115]
  MoveL 9980 to (509.44, 490.56, 18.7) mm, rotated rx 0 ry 90 rz 0 deg; joints [-10.972, -28.116, 110.809, -15.016, -82.078, 51.116]
  Set speed (120.0 mm/s)
  MoveL 9981 to (503.23, 493.33, 18.7) mm, rotated rx 0 ry 90 rz 0 deg; joints [-11.336, -28.228, 111.492, -15.363, -82.64, 51.009]
  Set speed (30.0 mm/s)
  Call Extruder(0.109)
  MoveL 9982 to (500.58, 490.68, 18.7) mm, rotated rx 0 ry 90 rz 0 deg; joints [-11.141, -28.289, 111.872, -15.156, -82.942, 50.903]
  Set speed (120.0 mm/s)
  MoveL 9983 to (499.42, 490.68, 18.7) mm, rotated rx 0 ry 90 rz 0 deg; joints [-11.163, -28.311, 112.011, -15.174, -83.056, 50.874]
  Set speed (30.0 mm/s)
  MoveL 9984 to (496.77, 493.33, 18.7) mm, rotated rx 0 ry 90 rz 0 deg; joints [-11.456, -28.35, 112.264, -15.462, -83.27, 50.848]
  MoveL 9985 to (496.65, 493.45, 18.7) mm, rotated rx 0 ry 90 rz 0 deg; joints [-11.47, -28.352, 112.276, -15.476, -83.28, 50.847]
  Set speed (120.0 mm/s)
  MoveL 9986 to (504.54, 493.58, 18.7) mm, rotated rx 0 ry 90 rz 0 deg; joints [-11.335, -28.202, 111.328, -15.367, -82.507, 51.046]
  Set speed (1000.0 mm/s)
  MoveL 9987 to (504.54, 495.95, 18.7) mm, rotated rx 0 ry 90 rz 0 deg; joints [-11.552, -28.192, 111.27, -15.587, -82.468, 51.084]
  Set speed (1000.0 mm/s)
  MoveL 9988 to (501.11, 498.89, 18.7) mm, rotated rx 0 ry 90 rz 0 deg; joints [-11.886, -28.247, 111.609, -15.913, -82.752, 51.045]
  Set speed (30.0 mm/s)
  Call Extruder(0.111)
  MoveL 9989 to (503.8, 496.2, 18.7) mm, rotated rx 0 ry 90 rz 0 deg; joints [-11.588, -28.206, 111.353, -15.621, -82.536, 51.069]
  MoveL 9990 to (503.92, 496.08, 18.7) mm, rotated rx 0 ry 90 rz 0 deg; joints [-11.575, -28.204, 111.342, -15.608, -82.526, 51.07]
  Set speed (120.0 mm/s)
  MoveL 9991 to (504.54, 493.58, 18.7) mm, rotated rx 0 ry 90 rz 0 deg; joints [-11.335, -28.202, 111.328, -15.367, -82.507, 51.046]
  Set speed (1000.0 mm/s)
  MoveL 9992 to (495.89, 493.58, 18.7) mm, rotated rx 0 ry 90 rz 0 deg; joints [-11.496, -28.365, 112.362, -15.5, -83.352, 50.83]
  Set speed (1000.0 mm/s)
  MoveL 9993 to (498.94, 501.06, 18.7) mm, rotated rx 0 ry 90 rz 0 deg; joints [-12.126, -28.28, 111.813, -16.15, -82.924, 51.023]
  Set speed (30.0 mm/s)
  Call Extruder(0.126)
  MoveL 9994 to (495.87, 504.12, 18.7) mm, rotated rx 0 ry 90 rz 0 deg; joints [-12.469, -28.324, 112.098, -16.487, -83.166, 50.992]
  MoveL 9995 to (495.75, 504.25, 18.7) mm, rotated rx 0 ry 90 rz 0 deg; joints [-12.483, -28.326, 112.11, -16.5, -83.175, 50.991]
  Set speed (120.0 mm/s)
  MoveL 9996 to (495.98, 506.75, 18.7) mm, rotated rx 0 ry 90 rz 0 deg; joints [-12.708, -28.312, 112.016, -16.729, -83.107, 51.037]
  Set speed (1000.0 mm/s)
  MoveL 9997 to (504.36, 506.75, 18.7) mm, rotated rx 0 ry 90 rz 0 deg; joints [-12.537, -28.15, 111.016, -16.588, -82.297, 51.26]
  Set speed (1000.0 mm/s)
  MoveL 9998 to (503.43, 503.43, 18.7) mm, rotated rx 0 ry 90 rz 0 deg; joints [-12.254, -28.183, 111.215, -16.296, -82.447, 51.179]
  Set speed (30.0 mm/s)
  Call Extruder(0.243)
  MoveL 9999 to (509.32, 509.32, 18.7) mm, rotated rx 0 ry 90 rz 0 deg; joints [-12.669, -28.037, 110.35, -16.743, -81.773, 51.437]
  MoveL 10000 to (509.44, 509.44, 18.7) mm, rotated rx 0 ry 90 rz 0 deg; joints [-12.677, -28.034, 110.332, -16.752, -81.759, 51.442]
  Set speed (120.0 mm/s)
  MoveL 10001 to (495.98, 506.75, 18.7) mm, rotated rx 0 ry 90 rz 0 deg; joints [-12.708, -28.312, 112.016, -16.729, -83.107, 51.037]
  Set speed (1000.0 mm/s)
  MoveL 10002 to (495.94, 504.33, 18.7) mm, rotated rx 0 ry 90 rz 0 deg; joints [-12.487, -28.322, 112.085, -16.505, -83.156, 50.997]
  Set speed (1000.0 mm/s)
  MoveL 10003 to (496.01, 504.41, 18.7) mm, rotated rx 0 ry 90 rz 0 deg; joints [-12.492, -28.321, 112.075, -16.511, -83.148, 51]
  Set speed (15.0 mm/s)
  Call Extruder(0.067)
  MoveL 10004 to (496.01, 506.72, 18.7) mm, rotated rx 0 ry 90 rz 0 deg; joints [-12.705, -28.311, 112.014, -16.726, -83.105, 51.037]
  Call Extruder(0.242)
  MoveL 10005 to (504.33, 506.72, 18.7) mm, rotated rx 0 ry 90 rz 0 deg; joints [-12.535, -28.151, 111.02, -16.586, -82.301, 51.259]
  Call Extruder(0.027)
  MoveL 10006 to (504.33, 505.8, 18.7) mm, rotated rx 0 ry 90 rz 0 deg; joints [-12.452, -28.155, 111.045, -16.501, -82.317, 51.243]
  Call Extruder(0.306)
  MoveL 10007 to (499.53, 496.43, 18.7) mm, rotated rx 0 ry 90 rz 0 deg; joints [-11.69, -28.287, 111.859, -15.709, -82.948, 50.965]
  Call Extruder(0.017)
  MoveL 10008 to (499.27, 495.92, 18.7) mm, rotated rx 0 ry 90 rz 0 deg; joints [-11.648, -28.294, 111.903, -15.666, -82.982, 50.951]
  Call Extruder(0.010)
  MoveL 10009 to (499.84, 495.92, 18.7) mm, rotated rx 0 ry 90 rz 0 deg; joints [-11.637, -28.283, 111.834, -15.657, -82.926, 50.965]
  Call Extruder(0.000)
  MoveL 10010 to (499.84, 495.92, 18.7) mm, rotated rx 0 ry 90 rz 0 deg; joints [-11.637, -28.283, 111.834, -15.657, -82.926, 50.965]
  Call Extruder(0.136)
  MoveL 10011 to (504.51, 495.92, 18.7) mm, rotated rx 0 ry 90 rz 0 deg; joints [-11.55, -28.193, 111.275, -15.584, -82.471, 51.083]
  Call Extruder(0.067)
  MoveL 10012 to (504.51, 493.61, 18.7) mm, rotated rx 0 ry 90 rz 0 deg; joints [-11.338, -28.202, 111.331, -15.37, -82.51, 51.045]
  Call Extruder(0.250)
  MoveL 10013 to (495.92, 493.61, 18.7) mm, rotated rx 0 ry 90 rz 0 deg; joints [-11.498, -28.364, 112.358, -15.502, -83.348, 50.831]
  Call Extruder(0.027)
  MoveL 10014 to (495.92, 494.52, 18.7) mm, rotated rx 0 ry 90 rz 0 deg; joints [-11.583, -28.361, 112.336, -15.588, -83.333, 50.844]
  Call Extruder(0.306)
  MoveL 10015 to (500.7, 503.9, 18.7) mm, rotated rx 0 ry 90 rz 0 deg; joints [-12.351, -28.234, 111.529, -16.384, -82.702, 51.116]
  Call Extruder(0.017)
  MoveL 10016 to (500.96, 504.41, 18.7) mm, rotated rx 0 ry 90 rz 0 deg; joints [-12.392, -28.227, 111.484, -16.427, -82.668, 51.131]
  Call Extruder(0.010)
  MoveL 10017 to (500.39, 504.41, 18.7) mm, rotated rx 0 ry 90 rz 0 deg; joints [-12.404, -28.238, 111.552, -16.437, -82.723, 51.116]
  Call Extruder(0.000)
  MoveL 10018 to (500.39, 504.41, 18.7) mm, rotated rx 0 ry 90 rz 0 deg; joints [-12.404, -28.238, 111.553, -16.437, -82.723, 51.116]
  Call Extruder(0.128)
  MoveL 10019 to (496.01, 504.41, 18.7) mm, rotated rx 0 ry 90 rz 0 deg; joints [-12.492, -28.321, 112.075, -16.511, -83.148, 51]
  Set speed (120.0 mm/s)
  MoveL 10020 to (496.01, 504.81, 18.7) mm, rotated rx 0 ry 90 rz 0 deg; joints [-12.529, -28.319, 112.065, -16.548, -83.14, 51.006]
  Set speed (1000.0 mm/s)
  MoveL 10021 to (495.91, 504.81, 18.7) mm, rotated rx 0 ry 90 rz 0 deg; joints [-12.531, -28.321, 112.077, -16.55, -83.15, 51.004]
  Set speed (1000.0 mm/s)
  MoveL 10022 to (490.47, 509.53, 18.7) mm, rotated rx 0 ry 90 rz 0 deg; joints [-13.08, -28.4, 112.594, -17.087, -83.586, 50.932]
  Set speed (1000.0 mm/s)
  MoveL 10023 to (490.4, 509.6, 18.7) mm, rotated rx 0 ry 90 rz 0 deg; joints [-13.088, -28.401, 112.6, -17.095, -83.591, 50.931]
  Set speed (15.0 mm/s)
  Call Extruder(0.559)
  MoveL 10024 to (490.4, 490.4, 18.7) mm, rotated rx 0 ry 90 rz 0 deg; joints [-11.303, -28.473, 113.091, -15.288, -83.945, 50.645]
  MoveL 10025 to (509.6, 490.4, 18.7) mm, rotated rx 0 ry 90 rz 0 deg; joints [-10.955, -28.113, 110.794, -14.999, -82.065, 51.118]
  MoveL 10026 to (509.6, 509.6, 18.7) mm, rotated rx 0 ry 90 rz 0 deg; joints [-12.688, -28.03, 110.308, -16.764, -81.74, 51.449]
  MoveL 10027 to (490.4, 509.6, 18.7) mm, rotated rx 0 ry 90 rz 0 deg; joints [-13.088, -28.401, 112.6, -17.095, -83.591, 50.931]
  Set speed (120.0 mm/s)
  MoveL 10028 to (490.4, 509.2, 18.7) mm, rotated rx 0 ry 90 rz 0 deg; joints [-13.051, -28.403, 112.611, -17.058, -83.599, 50.924]
  Set speed (1000.0 mm/s)
  MoveL 10029 to (491.1, 508.9, 18.7) mm, rotated rx 0 ry 90 rz 0 deg; joints [-13.008, -28.391, 112.536, -17.017, -83.537, 50.939]
  Set speed (1000.0 mm/s)
  MoveL 10030 to (490.68, 490.68, 18.7) mm, rotated rx 0 ry 90 rz 0 deg; joints [-11.324, -28.468, 113.051, -15.31, -83.913, 50.656]
  Set speed (1000.0 mm/s)
  MoveL 10031 to (490.68, 490.68, 18.8) mm, rotated rx 0 ry 90 rz 0 deg; joints [-11.324, -28.478, 113.056, -15.31, -83.907, 50.658]
  Set speed (30.0 mm/s)
  Call Extruder(0.249)
  MoveL 10032 to (496.74, 496.74, 18.8) mm, rotated rx 0 ry 90 rz 0 deg; joints [-11.772, -28.348, 112.19, -15.782, -83.209, 50.9]
  MoveL 10033 to (496.86, 496.86, 18.8) mm, rotated rx 0 ry 90 rz 0 deg; joints [-11.781, -28.346, 112.172, -15.792, -83.195, 50.905]
  Set speed (120.0 mm/s)
  MoveL 10034 to (495.64, 494.46, 18.8) mm, rotated rx 0 ry 90 rz 0 deg; joints [-11.582, -28.377, 112.376, -15.587, -83.356, 50.838]
  Set speed (30.0 mm/s)
  Call Extruder(0.204)
  MoveL 10035 to (490.68, 499.42, 18.8) mm, rotated rx 0 ry 90 rz 0 deg; joints [-12.139, -28.447, 112.841, -16.134, -83.752, 50.784]
  Set speed (120.0 mm/s)
  MoveL 10036 to (490.68, 500.58, 18.8) mm, rotated rx 0 ry 90 rz 0 deg; joints [-12.247, -28.442, 112.812, -16.244, -83.73, 50.801]
  Set speed (30.0 mm/s)
  Call Extruder(0.208)
  MoveL 10037 to (495.73, 505.63, 18.8) mm, rotated rx 0 ry 90 rz 0 deg; joints [-12.61, -28.332, 112.081, -16.629, -83.147, 51.014]
  Set speed (120.0 mm/s)
  MoveL 10038 to (495.72, 504.27, 18.8) mm, rotated rx 0 ry 90 rz 0 deg; joints [-12.486, -28.337, 112.117, -16.503, -83.172, 50.992]
  Set speed (30.0 mm/s)
  Call Extruder(0.208)
  MoveL 10039 to (490.68, 509.32, 18.8) mm, rotated rx 0 ry 90 rz 0 deg; joints [-13.056, -28.408, 112.58, -17.064, -83.564, 50.936]
  MoveL 10040 to (490.56, 509.44, 18.8) mm, rotated rx 0 ry 90 rz 0 deg; joints [-13.07, -28.41, 112.591, -17.078, -83.574, 50.934]
  Set speed (120.0 mm/s)
  MoveL 10041 to (497.1, 507, 18.8) mm, rotated rx 0 ry 90 rz 0 deg; joints [-12.708, -28.3, 111.882, -16.733, -82.989, 51.073]
  Set speed (30.0 mm/s)
  Call Extruder(0.096)
  MoveL 10042 to (499.42, 509.32, 18.8) mm, rotated rx 0 ry 90 rz 0 deg; joints [-12.872, -28.246, 111.542, -16.909, -82.721, 51.174]
  Set speed (120.0 mm/s)
  MoveL 10043 to (500.58, 509.32, 18.8) mm, rotated rx 0 ry 90 rz 0 deg; joints [-12.847, -28.224, 111.404, -16.889, -82.609, 51.205]
  Set speed (30.0 mm/s)
  Call Extruder(0.096)
  MoveL 10044 to (502.9, 507, 18.8) mm, rotated rx 0 ry 90 rz 0 deg; joints [-12.589, -28.189, 111.189, -16.635, -82.428, 51.228]
  MoveL 10045 to (503.02, 506.87, 18.8) mm, rotated rx 0 ry 90 rz 0 deg; joints [-12.575, -28.187, 111.177, -16.622, -82.418, 51.229]
  Set speed (120.0 mm/s)
  MoveL 10046 to (504.46, 505.44, 18.8) mm, rotated rx 0 ry 90 rz 0 deg; joints [-12.416, -28.164, 111.044, -16.466, -82.306, 51.242]
  Set speed (30.0 mm/s)
  Call Extruder(0.200)
  MoveL 10047 to (509.32, 500.58, 18.8) mm, rotated rx 0 ry 90 rz 0 deg; joints [-11.882, -28.087, 110.584, -15.941, -81.92, 51.283]
  Set speed (120.0 mm/s)
  MoveL 10048 to (509.32, 499.42, 18.8) mm, rotated rx 0 ry 90 rz 0 deg; joints [-11.777, -28.092, 110.614, -15.835, -81.94, 51.263]
  Set speed (30.0 mm/s)
  Call Extruder(0.186)
  MoveL 10049 to (504.79, 494.89, 18.8) mm, rotated rx 0 ry 90 rz 0 deg; joints [-11.45, -28.202, 111.271, -15.485, -82.456, 51.074]
  Set speed (120.0 mm/s)
  MoveL 10050 to (504.79, 495.21, 18.8) mm, rotated rx 0 ry 90 rz 0 deg; joints [-11.479, -28.201, 111.263, -15.514, -82.451, 51.08]
  Set speed (30.0 mm/s)
  Call Extruder(0.186)
  MoveL 10051 to (509.32, 490.68, 18.8) mm, rotated rx 0 ry 90 rz 0 deg; joints [-10.985, -28.128, 110.826, -15.029, -82.083, 51.117]
  MoveL 10052 to (509.44, 490.56, 18.8) mm, rotated rx 0 ry 90 rz 0 deg; joints [-10.972, -28.126, 110.814, -15.016, -82.073, 51.118]
  Set speed (120.0 mm/s)
  MoveL 10053 to (503.23, 493.33, 18.8) mm, rotated rx 0 ry 90 rz 0 deg; joints [-11.336, -28.239, 111.497, -15.363, -82.635, 51.011]
  Set speed (30.0 mm/s)
  Call Extruder(0.109)
  MoveL 10054 to (500.58, 490.68, 18.8) mm, rotated rx 0 ry 90 rz 0 deg; joints [-11.141, -28.3, 111.877, -15.156, -82.937, 50.904]
  Set speed (120.0 mm/s)
  MoveL 10055 to (499.42, 490.68, 18.8) mm, rotated rx 0 ry 90 rz 0 deg; joints [-11.163, -28.321, 112.016, -15.174, -83.05, 50.876]
  Set speed (30.0 mm/s)
  MoveL 10056 to (496.77, 493.33, 18.8) mm, rotated rx 0 ry 90 rz 0 deg; joints [-11.456, -28.361, 112.269, -15.463, -83.265, 50.849]
  MoveL 10057 to (496.65, 493.45, 18.8) mm, rotated rx 0 ry 90 rz 0 deg; joints [-11.47, -28.362, 112.281, -15.476, -83.275, 50.848]
  Set speed (120.0 mm/s)
  MoveL 10058 to (504.54, 493.58, 18.8) mm, rotated rx 0 ry 90 rz 0 deg; joints [-11.335, -28.212, 111.333, -15.367, -82.502, 51.047]
  Set speed (1000.0 mm/s)
  MoveL 10059 to (504.54, 495.95, 18.8) mm, rotated rx 0 ry 90 rz 0 deg; joints [-11.552, -28.203, 111.276, -15.587, -82.463, 51.085]
  Set speed (1000.0 mm/s)
  MoveL 10060 to (501.11, 498.89, 18.8) mm, rotated rx 0 ry 90 rz 0 deg; joints [-11.886, -28.258, 111.614, -15.913, -82.746, 51.046]
  Set speed (30.0 mm/s)
  Call Extruder(0.111)
  MoveL 10061 to (503.8, 496.2, 18.8) mm, rotated rx 0 ry 90 rz 0 deg; joints [-11.588, -28.216, 111.358, -15.622, -82.531, 51.071]
  MoveL 10062 to (503.92, 496.08, 18.8) mm, rotated rx 0 ry 90 rz 0 deg; joints [-11.575, -28.214, 111.347, -15.608, -82.521, 51.072]
  Set speed (120.0 mm/s)
  MoveL 10063 to (504.54, 493.58, 18.8) mm, rotated rx 0 ry 90 rz 0 deg; joints [-11.335, -28.212, 111.333, -15.367, -82.502, 51.047]
  Set speed (1000.0 mm/s)
  MoveL 10064 to (495.89, 493.58, 18.8) mm, rotated rx 0 ry 90 rz 0 deg; joints [-11.496, -28.376, 112.367, -15.5, -83.346, 50.831]
  Set speed (1000.0 mm/s)
  MoveL 10065 to (498.94, 501.06, 18.8) mm, rotated rx 0 ry 90 rz 0 deg; joints [-12.126, -28.29, 111.818, -16.15, -82.919, 51.025]
  Set speed (30.0 mm/s)
  Call Extruder(0.126)
  MoveL 10066 to (495.87, 504.12, 18.8) mm, rotated rx 0 ry 90 rz 0 deg; joints [-12.469, -28.335, 112.103, -16.487, -83.16, 50.994]
  MoveL 10067 to (495.75, 504.25, 18.8) mm, rotated rx 0 ry 90 rz 0 deg; joints [-12.483, -28.337, 112.115, -16.5, -83.17, 50.992]
  Set speed (120.0 mm/s)
  MoveL 10068 to (495.98, 506.75, 18.8) mm, rotated rx 0 ry 90 rz 0 deg; joints [-12.708, -28.322, 112.021, -16.729, -83.101, 51.039]
  Set speed (1000.0 mm/s)
  MoveL 10069 to (504.36, 506.75, 18.8) mm, rotated rx 0 ry 90 rz 0 deg; joints [-12.537, -28.161, 111.021, -16.588, -82.292, 51.262]
  Set speed (1000.0 mm/s)
  MoveL 10070 to (503.43, 503.43, 18.8) mm, rotated rx 0 ry 90 rz 0 deg; joints [-12.254, -28.194, 111.22, -16.297, -82.441, 51.181]
  Set speed (30.0 mm/s)
  Call Extruder(0.243)
  MoveL 10071 to (509.32, 509.32, 18.8) mm, rotated rx 0 ry 90 rz 0 deg; joints [-12.669, -28.047, 110.355, -16.743, -81.767, 51.438]
  MoveL 10072 to (509.44, 509.44, 18.8) mm, rotated rx 0 ry 90 rz 0 deg; joints [-12.677, -28.044, 110.337, -16.753, -81.753, 51.444]
  Set speed (120.0 mm/s)
  MoveL 10073 to (495.98, 506.75, 18.8) mm, rotated rx 0 ry 90 rz 0 deg; joints [-12.708, -28.322, 112.021, -16.729, -83.101, 51.039]
  Set speed (1000.0 mm/s)
  MoveL 10074 to (495.94, 504.33, 18.8) mm, rotated rx 0 ry 90 rz 0 deg; joints [-12.487, -28.333, 112.091, -16.505, -83.15, 50.999]
  Set speed (1000.0 mm/s)
  MoveL 10075 to (496.01, 504.4, 18.8) mm, rotated rx 0 ry 90 rz 0 deg; joints [-12.492, -28.331, 112.08, -16.511, -83.142, 51.002]
  Set speed (15.0 mm/s)
  Call Extruder(0.067)
  MoveL 10076 to (496.01, 506.72, 18.8) mm, rotated rx 0 ry 90 rz 0 deg; joints [-12.705, -28.322, 112.019, -16.726, -83.099, 51.039]
  Call Extruder(0.242)
  MoveL 10077 to (504.33, 506.72, 18.8) mm, rotated rx 0 ry 90 rz 0 deg; joints [-12.535, -28.161, 111.025, -16.586, -82.295, 51.26]
  Call Extruder(0.027)
  MoveL 10078 to (504.33, 505.8, 18.8) mm, rotated rx 0 ry 90 rz 0 deg; joints [-12.452, -28.165, 111.05, -16.501, -82.312, 51.245]
  Call Extruder(0.306)
  MoveL 10079 to (499.53, 496.43, 18.8) mm, rotated rx 0 ry 90 rz 0 deg; joints [-11.69, -28.298, 111.864, -15.709, -82.942, 50.967]
  Call Extruder(0.017)
  MoveL 10080 to (499.27, 495.92, 18.8) mm, rotated rx 0 ry 90 rz 0 deg; joints [-11.648, -28.304, 111.908, -15.666, -82.977, 50.952]
  Call Extruder(0.010)
  MoveL 10081 to (499.84, 495.92, 18.8) mm, rotated rx 0 ry 90 rz 0 deg; joints [-11.637, -28.294, 111.839, -15.657, -82.921, 50.967]
  Call Extruder(0.000)
  MoveL 10082 to (499.84, 495.92, 18.8) mm, rotated rx 0 ry 90 rz 0 deg; joints [-11.637, -28.294, 111.839, -15.657, -82.921, 50.967]
  Call Extruder(0.136)
  MoveL 10083 to (504.51, 495.92, 18.8) mm, rotated rx 0 ry 90 rz 0 deg; joints [-11.55, -28.203, 111.28, -15.585, -82.466, 51.084]
  Call Extruder(0.067)
  MoveL 10084 to (504.51, 493.61, 18.8) mm, rotated rx 0 ry 90 rz 0 deg; joints [-11.338, -28.213, 111.336, -15.37, -82.504, 51.047]
  Call Extruder(0.250)
  MoveL 10085 to (495.92, 493.61, 18.8) mm, rotated rx 0 ry 90 rz 0 deg; joints [-11.498, -28.375, 112.363, -15.502, -83.343, 50.832]
  Call Extruder(0.027)
  MoveL 10086 to (495.92, 494.52, 18.8) mm, rotated rx 0 ry 90 rz 0 deg; joints [-11.583, -28.372, 112.341, -15.588, -83.327, 50.846]
  Call Extruder(0.306)
  MoveL 10087 to (500.7, 503.9, 18.8) mm, rotated rx 0 ry 90 rz 0 deg; joints [-12.351, -28.245, 111.534, -16.385, -82.697, 51.117]
  Call Extruder(0.017)
  MoveL 10088 to (500.96, 504.41, 18.8) mm, rotated rx 0 ry 90 rz 0 deg; joints [-12.392, -28.238, 111.489, -16.428, -82.662, 51.133]
  Call Extruder(0.010)
  MoveL 10089 to (500.39, 504.41, 18.8) mm, rotated rx 0 ry 90 rz 0 deg; joints [-12.404, -28.249, 111.557, -16.437, -82.717, 51.118]
  Call Extruder(0.000)
  MoveL 10090 to (500.39, 504.41, 18.8) mm, rotated rx 0 ry 90 rz 0 deg; joints [-12.404, -28.249, 111.558, -16.437, -82.718, 51.118]
  Call Extruder(0.128)
  MoveL 10091 to (496.01, 504.4, 18.8) mm, rotated rx 0 ry 90 rz 0 deg; joints [-12.492, -28.331, 112.08, -16.511, -83.142, 51.002]
  Set speed (120.0 mm/s)
  MoveL 10092 to (496.01, 504.81, 18.8) mm, rotated rx 0 ry 90 rz 0 deg; joints [-12.529, -28.33, 112.07, -16.548, -83.135, 51.008]
  Set speed (1000.0 mm/s)
  MoveL 10093 to (495.91, 504.8, 18.8) mm, rotated rx 0 ry 90 rz 0 deg; joints [-12.531, -28.332, 112.082, -16.55, -83.145, 51.005]
  Set speed (1000.0 mm/s)
  MoveL 10094 to (490.47, 509.53, 18.8) mm, rotated rx 0 ry 90 rz 0 deg; joints [-13.08, -28.411, 112.599, -17.087, -83.58, 50.933]
  Set speed (1000.0 mm/s)
  MoveL 10095 to (490.4, 509.6, 18.8) mm, rotated rx 0 ry 90 rz 0 deg; joints [-13.088, -28.412, 112.605, -17.095, -83.586, 50.932]
  Set speed (15.0 mm/s)
  Call Extruder(0.559)
  MoveL 10096 to (490.4, 490.4, 18.8) mm, rotated rx 0 ry 90 rz 0 deg; joints [-11.303, -28.484, 113.096, -15.288, -83.939, 50.647]
  MoveL 10097 to (509.6, 490.4, 18.8) mm, rotated rx 0 ry 90 rz 0 deg; joints [-10.955, -28.123, 110.799, -14.999, -82.06, 51.119]
  MoveL 10098 to (509.6, 509.6, 18.8) mm, rotated rx 0 ry 90 rz 0 deg; joints [-12.688, -28.04, 110.314, -16.764, -81.735, 51.451]
  MoveL 10099 to (490.4, 509.6, 18.8) mm, rotated rx 0 ry 90 rz 0 deg; joints [-13.088, -28.412, 112.605, -17.095, -83.586, 50.932]
  Set speed (120.0 mm/s)
  MoveL 10100 to (490.4, 509.2, 18.8) mm, rotated rx 0 ry 90 rz 0 deg; joints [-13.051, -28.413, 112.616, -17.058, -83.594, 50.926]
  Set speed (1000.0 mm/s)
  MoveL 10101 to (491.1, 508.9, 18.8) mm, rotated rx 0 ry 90 rz 0 deg; joints [-13.008, -28.402, 112.541, -17.017, -83.532, 50.941]
  Set speed (1000.0 mm/s)
  MoveL 10102 to (490.68, 490.68, 18.8) mm, rotated rx 0 ry 90 rz 0 deg; joints [-11.324, -28.478, 113.056, -15.31, -83.907, 50.658]
  Set speed (1000.0 mm/s)
  MoveL 10103 to (490.68, 490.68, 18.9) mm, rotated rx 0 ry 90 rz 0 deg; joints [-11.324, -28.489, 113.061, -15.31, -83.902, 50.659]
  Set speed (30.0 mm/s)
  Call Extruder(0.249)
  MoveL 10104 to (496.74, 496.74, 18.9) mm, rotated rx 0 ry 90 rz 0 deg; joints [-11.772, -28.359, 112.195, -15.783, -83.204, 50.902]
  MoveL 10105 to (496.86, 496.86, 18.9) mm, rotated rx 0 ry 90 rz 0 deg; joints [-11.781, -28.356, 112.177, -15.792, -83.19, 50.907]
  Set speed (120.0 mm/s)
  MoveL 10106 to (495.64, 494.46, 18.9) mm, rotated rx 0 ry 90 rz 0 deg; joints [-11.582, -28.388, 112.381, -15.587, -83.351, 50.839]
  Set speed (30.0 mm/s)
  Call Extruder(0.204)
  MoveL 10107 to (490.68, 499.42, 18.9) mm, rotated rx 0 ry 90 rz 0 deg; joints [-12.139, -28.457, 112.846, -16.135, -83.746, 50.785]
  Set speed (120.0 mm/s)
  MoveL 10108 to (490.68, 500.58, 18.9) mm, rotated rx 0 ry 90 rz 0 deg; joints [-12.247, -28.453, 112.817, -16.244, -83.725, 50.802]
  Set speed (30.0 mm/s)
  Call Extruder(0.208)
  MoveL 10109 to (495.73, 505.63, 18.9) mm, rotated rx 0 ry 90 rz 0 deg; joints [-12.61, -28.342, 112.086, -16.63, -83.141, 51.015]
  Set speed (120.0 mm/s)
  MoveL 10110 to (495.73, 504.27, 18.9) mm, rotated rx 0 ry 90 rz 0 deg; joints [-12.486, -28.348, 112.122, -16.503, -83.167, 50.994]
  Set speed (30.0 mm/s)
  Call Extruder(0.208)
  MoveL 10111 to (490.68, 509.32, 18.9) mm, rotated rx 0 ry 90 rz 0 deg; joints [-13.056, -28.419, 112.585, -17.064, -83.559, 50.937]
  MoveL 10112 to (490.56, 509.44, 18.9) mm, rotated rx 0 ry 90 rz 0 deg; joints [-13.07, -28.42, 112.596, -17.078, -83.569, 50.936]
  Set speed (120.0 mm/s)
  MoveL 10113 to (497.1, 507, 18.9) mm, rotated rx 0 ry 90 rz 0 deg; joints [-12.708, -28.311, 111.887, -16.734, -82.983, 51.074]
  Set speed (30.0 mm/s)
  Call Extruder(0.096)
  MoveL 10114 to (499.42, 509.32, 18.9) mm, rotated rx 0 ry 90 rz 0 deg; joints [-12.872, -28.257, 111.547, -16.909, -82.716, 51.176]
  Set speed (120.0 mm/s)
  MoveL 10115 to (500.58, 509.32, 18.9) mm, rotated rx 0 ry 90 rz 0 deg; joints [-12.847, -28.234, 111.409, -16.889, -82.604, 51.207]
  Set speed (30.0 mm/s)
  Call Extruder(0.096)
  MoveL 10116 to (502.9, 507, 18.9) mm, rotated rx 0 ry 90 rz 0 deg; joints [-12.589, -28.199, 111.194, -16.635, -82.423, 51.229]
  MoveL 10117 to (503.02, 506.87, 18.9) mm, rotated rx 0 ry 90 rz 0 deg; joints [-12.575, -28.197, 111.182, -16.622, -82.413, 51.23]
  Set speed (120.0 mm/s)
  MoveL 10118 to (504.46, 505.44, 18.9) mm, rotated rx 0 ry 90 rz 0 deg; joints [-12.416, -28.175, 111.049, -16.466, -82.301, 51.243]
  Set speed (30.0 mm/s)
  Call Extruder(0.200)
  MoveL 10119 to (509.32, 500.58, 18.9) mm, rotated rx 0 ry 90 rz 0 deg; joints [-11.882, -28.097, 110.589, -15.942, -81.915, 51.285]
  Set speed (120.0 mm/s)
  MoveL 10120 to (509.32, 499.42, 18.9) mm, rotated rx 0 ry 90 rz 0 deg; joints [-11.777, -28.102, 110.619, -15.835, -81.935, 51.265]
  Set speed (30.0 mm/s)
  Call Extruder(0.186)
  MoveL 10121 to (504.79, 494.89, 18.9) mm, rotated rx 0 ry 90 rz 0 deg; joints [-11.45, -28.213, 111.276, -15.485, -82.451, 51.076]
  Set speed (120.0 mm/s)
  MoveL 10122 to (504.79, 495.21, 18.9) mm, rotated rx 0 ry 90 rz 0 deg; joints [-11.479, -28.211, 111.269, -15.515, -82.445, 51.081]
  Set speed (30.0 mm/s)
  Call Extruder(0.186)
  MoveL 10123 to (509.32, 490.68, 18.9) mm, rotated rx 0 ry 90 rz 0 deg; joints [-10.985, -28.139, 110.831, -15.029, -82.078, 51.118]
  MoveL 10124 to (509.44, 490.56, 18.9) mm, rotated rx 0 ry 90 rz 0 deg; joints [-10.972, -28.137, 110.819, -15.016, -82.068, 51.119]
  Set speed (120.0 mm/s)
  MoveL 10125 to (503.23, 493.33, 18.9) mm, rotated rx 0 ry 90 rz 0 deg; joints [-11.336, -28.249, 111.502, -15.364, -82.629, 51.012]
  Set speed (30.0 mm/s)
  Call Extruder(0.109)
  MoveL 10126 to (500.58, 490.68, 18.9) mm, rotated rx 0 ry 90 rz 0 deg; joints [-11.141, -28.31, 111.882, -15.157, -82.932, 50.906]
  Set speed (120.0 mm/s)
  MoveL 10127 to (499.42, 490.68, 18.9) mm, rotated rx 0 ry 90 rz 0 deg; joints [-11.163, -28.332, 112.021, -15.174, -83.045, 50.877]
  Set speed (30.0 mm/s)
  MoveL 10128 to (496.77, 493.33, 18.9) mm, rotated rx 0 ry 90 rz 0 deg; joints [-11.456, -28.371, 112.274, -15.463, -83.259, 50.851]
  MoveL 10129 to (496.65, 493.45, 18.9) mm, rotated rx 0 ry 90 rz 0 deg; joints [-11.47, -28.373, 112.286, -15.476, -83.269, 50.85]
  Set speed (120.0 mm/s)
  MoveL 10130 to (504.54, 493.58, 18.9) mm, rotated rx 0 ry 90 rz 0 deg; joints [-11.335, -28.223, 111.338, -15.367, -82.497, 51.049]
